# B&R Automation Studio project Panasonic_LinkaKapacitorov_A2021040 (part 6)

#### Main.st - Init, cyclic, exit code
```iecst
PROGRAM _INIT
	(* Insert code here *)

END_PROGRAM

PROGRAM _CYCLIC

	//Meranie motohodin ionizátora Tajfun//

	Tajfun_Motohodiny.START:= Linka.OUT.IonJednotka_START;

	//Spustenie merania//
	IF Tajfun_Motohodiny.START THEN
		Tajfun_Motohodiny.Milisekundy:= Tajfun_Motohodiny.Milisekundy + 2;//Ak je v taskovej triede 2ms tak prirátaváme + 2//
	END_IF

	IF Tajfun_Motohodiny.Milisekundy >= 1000 THEN
		Tajfun_Motohodiny.Sekundy:= Tajfun_Motohodiny.Sekundy + 1;
		Tajfun_Motohodiny.Milisekundy:= 0;
	END_IF

	IF Tajfun_Motohodiny.Sekundy >= 60 THEN
		Tajfun_Motohodiny.Minuty:= Tajfun_Motohodiny.Minuty + 1;
		Tajfun_Motohodiny.Sekundy:= 0;
	END_IF

	IF Tajfun_Motohodiny.Minuty >= 60 THEN
		Tajfun_Motohodiny.Hodiny:= Tajfun_Motohodiny.Hodiny + 1;
		Tajfun_Motohodiny.CelkovyPocetHodin:= Tajfun_Motohodiny.CelkovyPocetHodin + 1;
		Tajfun_Motohodiny.Minuty:= 0;
	END_IF

	IF Tajfun_Motohodiny.Hodiny >= 24 THEN
		Tajfun_Motohodiny.Dny:= Tajfun_Motohodiny.Dny + 1;
		Tajfun_Motohodiny.Hodiny:= 0;
	END_IF

	//Reset merania//
	IF Tajfun_Motohodiny.RESET THEN
		Tajfun_Motohodiny.Milisekundy:= 0;
		Tajfun_Motohodiny.Sekundy:= 0;
		Tajfun_Motohodiny.Minuty:= 0;
		Tajfun_Motohodiny.Hodiny:= 0;
		Tajfun_Motohodiny.CelkovyPocetHodin:= 0;
		Tajfun_Motohodiny.Dny:= 0;
		Tajfun_Motohodiny.RESET:= FALSE;
	END_IF

	//Zobrazenie stavov filtrov ionizačnej jednotky//
	//0 - Stav filtrov ionizačnej jednotky je OK.
	//1 - Blíži sa termín výmeny filtrov ionizačnej jednotky !!!
	//2 - Nutná výmena filtrov ionizačnej jednotky !!!

	//Farby stavov filtrov//
	//0 - Sivá
	//1 - Zelená
	//2 - Oranžová
	//3 - Červená

	CasKontrolyFiltrov.IN:= Linka.OUT.IonJednotka_START;

	IF Safety.STAV.SafetyPLC_Nabehlo THEN
		IF CasKontrolyFiltrov.Q AND (NOT Linka.IN.IonJednotka_Error_Filter1_RJ1 OR NOT Linka.IN.IonJednotka_Error_Filter2_RJ1)THEN
			Linka.STAV.FiltreIonizacnejJednotkyZanesene:= TRUE;
			Vizu.IndexStavuFiltrov:= 2;
			Vizu.IndexFarbyStavuFiltrov:= 3;
		ELSIF Tajfun_Motohodiny.Dny >= RemPremenne.PocetDniDoVymenyFiltra THEN
			Linka.STAV.FiltreIonizacnejJednotkyZanesene:= TRUE;
			Vizu.IndexStavuFiltrov:= 2;
			Vizu.IndexFarbyStavuFiltrov:= 3;
		ELSIF Tajfun_Motohodiny.Dny >= RemPremenne.PocetDniDoVymenyFiltra - 7 THEN
			Vizu.IndexStavuFiltrov:= 1;
			Vizu.IndexFarbyStavuFiltrov:= 2;
		ELSE
			Vizu.IndexStavuFiltrov:= 0;
			Vizu.IndexFarbyStavuFiltrov:= 1;
		END_IF
	END_IF

	IF Linka.VymenaFiltrovPotvrdena THEN
		Linka.STAV.FiltreIonizacnejJednotkyZanesene:= FALSE;
		Tajfun_Motohodiny.RESET:= TRUE;
		Linka.VymenaFiltrovPotvrdena:= FALSE;
	END_IF

	CasKontrolyFiltrov.PT:= T#2s;
	CasKontrolyFiltrov();

END_PROGRAM

PROGRAM _EXIT
	(* Insert code here *)

END_PROGRAM
```

#### Variables.var - Local variables
```iecst
VAR
	CasKontrolyFiltrov : TON := (0);
END_VAR
```

### Program Logical/Program/TestKomunikacie (IEC)

#### Main.st - Init, cyclic, exit code
```iecst
PROGRAM _INIT
	(* Insert code here *)

END_PROGRAM

PROGRAM _CYCLIC

	//Volanie funkcie SequenceControl//
	SequenceControl(SC:= SC_Step);

	CASE SC_Step.Step OF

		0:
			SC_Step.StepName:='0 - Nulovanie';
			Cistenie_OK:= FALSE;
			Cistenie_NG:= FALSE;
			VytlacEtiketu:= FALSE;
			NalepenieEtikety_OK:= FALSE;
			NalepenieEikety_NG:= FALSE;
			KontrolaDMkodu_OK:= FALSE;
			KontrolaDMkodu_NG:= FALSE;
			KontrolaTextu_OK:= FALSE;
			KontrolaTextu_NG:= FALSE;
			KOM_Panasonic.Server_IN.DataForServer_READY:= FALSE;
			KOM_Panasonic.Server_IN.ProcessResult:= FALSE;
			KOM_Panasonic.Server_IN.CommandNumber:= 0;
			SC_Step.ResetStep:= TRUE;
			SC_Step.Step:= 1;

		1:
			IF Cistenie_OK THEN
				ZakaznickeCislo:= '';
				ReturnProcessName:= '';
				SC_Step.ResetStep:= TRUE;
				SC_Step.Step:= 10;
			ELSIF Cistenie_NG THEN
				ZakaznickeCislo:= '';
				ReturnProcessName:= '';
				SC_Step.ResetStep:= TRUE;
				SC_Step.Step:= 20;
			ELSIF VytlacEtiketu THEN
				ReturnProcessName:= '';
				SC_Step.ResetStep:= TRUE;
				SC_Step.Step:= 30;
			ELSIF NalepenieEtikety_OK THEN
				ReturnProcessName:= '';
				SC_Step.ResetStep:= TRUE;
				SC_Step.Step:= 40;
			ELSIF NalepenieEikety_NG THEN
				ReturnProcessName:= '';
				SC_Step.ResetStep:= TRUE;
				SC_Step.Step:= 50;
			ELSIF KontrolaDMkodu_OK THEN
				ReturnProcessName:= '';
				SC_Step.ResetStep:= TRUE;
				SC_Step.Step:= 60;
			ELSIF KontrolaDMkodu_NG THEN
				ReturnProcessName:= '';
				SC_Step.ResetStep:= TRUE;
				SC_Step.Step:= 70;
			ELSIF KontrolaTextu_OK THEN
				ReturnProcessName:= '';
				SC_Step.ResetStep:= TRUE;
				SC_Step.Step:= 80;
			ELSIF KontrolaTextu_NG THEN
				ReturnProcessName:= '';
				SC_Step.ResetStep:= TRUE;
				SC_Step.Step:= 90;
			END_IF

		10:
			SC_Step.StepName:='10 - Odoslanie - Stav cistenie OK';
			SC_Step.IdleTime.PT:= T#4s;
			SC_Step.AlarmTime.PT:= T#5s;

			KOM_Panasonic.Server_IN.NazovPaletky_RFID:= '10_CP1';
			KOM_Panasonic.Server_IN.SerialNumber_InternaEtiketa:= 'BD10020070300046ZZZZZZZB10BD1';
			KOM_Panasonic.Server_IN.Cislo_LOTU:= 'BS217210002';

			IF NOT KOM_Panasonic.Server_OUT.DataForPLC_READY THEN
				KOM_Panasonic.Server_IN.CommandNumber:= 10;
				KOM_Panasonic.Server_IN.ProcessResult:= TRUE;
				KOM_Panasonic.Server_IN.DataForServer_READY:= TRUE;
				SC_Step.ResetStep:= TRUE;
				SC_Step.Step:= 13;
			END_IF

		13:
			SC_Step.StepName:='13 - Odpoved servera';
			SC_Step.IdleTime.PT:= T#100ms;
			SC_Step.AlarmTime.PT:= T#5s;

			IF KOM_Panasonic.Server_OUT.DataForPLC_READY AND KOM_Panasonic.Server_OUT.LastCommandNumber = 10 THEN
				IF KOM_Panasonic.Server_OUT.ContinueToNextProcess THEN
					ZakaznickeCislo:= KOM_Panasonic.Server_OUT.SerialNumber_ZakaznickaEtiketa;
					KOM_Panasonic.Server_IN.DataForServer_READY:= FALSE;
					ReturnProcessName:= 'OK';
					SC_Step.ResetStep:= TRUE;
					SC_Step.Step:= 0;
				ELSIF NOT KOM_Panasonic.Server_OUT.ContinueToNextProcess THEN
					ReturnProcessName:= KOM_Panasonic.Server_OUT.ReturnProcessName;
					KOM_Panasonic.Server_IN.DataForServer_READY:= FALSE;
					SC_Step.ResetStep:= TRUE;
					SC_Step.Step:= 0;
				END_IF
			END_IF

		20:
			SC_Step.StepName:='20 - Odoslanie - Stav cistenie NG';
			SC_Step.IdleTime.PT:= T#4s;
			SC_Step.AlarmTime.PT:= T#5s;

			KOM_Panasonic.Server_IN.NazovPaletky_RFID:= '10_CP1';
			KOM_Panasonic.Server_IN.SerialNumber_InternaEtiketa:= 'BD10020070300046ZZZZZZZB10BD1';
			KOM_Panasonic.Server_IN.Cislo_LOTU:= 'BS217210002';

			IF NOT KOM_Panasonic.Server_OUT.DataForPLC_READY THEN
				KOM_Panasonic.Server_IN.CommandNumber:= 10;
				KOM_Panasonic.Server_IN.ProcessResult:= FALSE;
				KOM_Panasonic.Server_IN.DataForServer_READY:= TRUE;
				SC_Step.ResetStep:= TRUE;
				SC_Step.Step:= 23;
			END_IF

		23:
			SC_Step.StepName:='23 - Odpoved servera';
			SC_Step.IdleTime.PT:= T#100ms;
			SC_Step.AlarmTime.PT:= T#5s;

			IF KOM_Panasonic.Server_OUT.DataForPLC_READY AND KOM_Panasonic.Server_OUT.LastCommandNumber = 10 THEN
				IF KOM_Panasonic.Server_OUT.ContinueToNextProcess THEN
					ZakaznickeCislo:= KOM_Panasonic.Server_OUT.SerialNumber_ZakaznickaEtiketa;
					KOM_Panasonic.Server_IN.DataForServer_READY:= FALSE;
					ReturnProcessName:= 'OK';
					SC_Step.ResetStep:= TRUE;
					SC_Step.Step:= 0;
				ELSIF NOT KOM_Panasonic.Server_OUT.ContinueToNextProcess THEN
					ReturnProcessName:= KOM_Panasonic.Server_OUT.ReturnProcessName;
					KOM_Panasonic.Server_IN.DataForServer_READY:= FALSE;
					SC_Step.ResetStep:= TRUE;
					SC_Step.Step:= 0;
				END_IF
			END_IF

		30:
			SC_Step.StepName:='30 - Odoslanie - Vytlac etiketu';
			SC_Step.IdleTime.PT:= T#4s;
			SC_Step.AlarmTime.PT:= T#5s;

			KOM_Panasonic.Server_IN.NazovPaletky_RFID:= '10_CP1';
			KOM_Panasonic.Server_IN.SerialNumber_InternaEtiketa:= 'BD10020070300046ZZZZZZZB10BD1';
			KOM_Panasonic.Server_IN.Cislo_LOTU:= 'BS217210002';

			IF NOT KOM_Panasonic.Server_OUT.DataForPLC_READY THEN
				KOM_Panasonic.Server_IN.CommandNumber:= 20;
				KOM_Panasonic.Server_IN.ProcessResult:= TRUE;
				KOM_Panasonic.Server_IN.DataForServer_READY:= TRUE;
				SC_Step.ResetStep:= TRUE;
				SC_Step.Step:= 33;
			END_IF

		33:
			SC_Step.StepName:='33 - Odpoved servera';
			SC_Step.IdleTime.PT:= T#100ms;
			SC_Step.AlarmTime.PT:= T#5s;

			IF KOM_Panasonic.Server_OUT.DataForPLC_READY AND KOM_Panasonic.Server_OUT.LastCommandNumber = 20 THEN
				IF KOM_Panasonic.Server_OUT.ContinueToNextProcess THEN
					KOM_Panasonic.Server_IN.DataForServer_READY:= FALSE;
					ReturnProcessName:= 'OK';
					SC_Step.ResetStep:= TRUE;
					SC_Step.Step:= 0;
				ELSIF NOT KOM_Panasonic.Server_OUT.ContinueToNextProcess THEN
					ReturnProcessName:= KOM_Panasonic.Server_OUT.ReturnProcessName;
					KOM_Panasonic.Server_IN.DataForServer_READY:= FALSE;
					SC_Step.ResetStep:= TRUE;
					SC_Step.Step:= 0;
				END_IF
			END_IF

		40:
			SC_Step.StepName:='40 - Odoslanie - Stav nalepenie etikety OK';
			SC_Step.IdleTime.PT:= T#4s;
			SC_Step.AlarmTime.PT:= T#5s;

			KOM_Panasonic.Server_IN.NazovPaletky_RFID:= '10_CP1';
			KOM_Panasonic.Server_IN.SerialNumber_InternaEtiketa:= 'BD10020070300046ZZZZZZZB10BD1';
			KOM_Panasonic.Server_IN.Cislo_LOTU:= 'BS217210002';

			IF NOT KOM_Panasonic.Server_OUT.DataForPLC_READY THEN
				KOM_Panasonic.Server_IN.CommandNumber:= 30;
				KOM_Panasonic.Server_IN.ProcessResult:= TRUE;
				KOM_Panasonic.Server_IN.DataForServer_READY:= TRUE;
				SC_Step.ResetStep:= TRUE;
				SC_Step.Step:= 43;
			END_IF

		43:
			SC_Step.StepName:='43 - Odpoved servera';
			SC_Step.IdleTime.PT:= T#100ms;
			SC_Step.AlarmTime.PT:= T#5s;

			IF KOM_Panasonic.Server_OUT.DataForPLC_READY AND KOM_Panasonic.Server_OUT.LastCommandNumber = 30 THEN
				IF KOM_Panasonic.Server_OUT.ContinueToNextProcess THEN
					KOM_Panasonic.Server_IN.DataForServer_READY:= FALSE;
					ReturnProcessName:= 'OK';
					SC_Step.ResetStep:= TRUE;
					SC_Step.Step:= 0;
				ELSIF NOT KOM_Panasonic.Server_OUT.ContinueToNextProcess THEN
					ReturnProcessName:= KOM_Panasonic.Server_OUT.ReturnProcessName;
					KOM_Panasonic.Server_IN.DataForServer_READY:= FALSE;
					SC_Step.ResetStep:= TRUE;
					SC_Step.Step:= 0;
				END_IF
			END_IF

		50:
			SC_Step.StepName:='50 - Odoslanie - Stav nalepenie etikety NG';
			SC_Step.IdleTime.PT:= T#4s;
			SC_Step.AlarmTime.PT:= T#5s;

			KOM_Panasonic.Server_IN.NazovPaletky_RFID:= '10_CP1';
			KOM_Panasonic.Server_IN.SerialNumber_InternaEtiketa:= 'BD10020070300046ZZZZZZZB10BD1';
			KOM_Panasonic.Server_IN.Cislo_LOTU:= 'BS217210002';

			IF NOT KOM_Panasonic.Server_OUT.DataForPLC_READY THEN
				KOM_Panasonic.Server_IN.CommandNumber:= 30;
				KOM_Panasonic.Server_IN.ProcessResult:= FALSE;
				KOM_Panasonic.Server_IN.DataForServer_READY:= TRUE;
				SC_Step.ResetStep:= TRUE;
				SC_Step.Step:= 53;
			END_IF

		53:
			SC_Step.StepName:='53 - Odpoved servera';
			SC_Step.IdleTime.PT:= T#100ms;
			SC_Step.AlarmTime.PT:= T#5s;

			IF KOM_Panasonic.Server_OUT.DataForPLC_READY AND KOM_Panasonic.Server_OUT.LastCommandNumber = 30 THEN
				IF KOM_Panasonic.Server_OUT.ContinueToNextProcess THEN
					KOM_Panasonic.Server_IN.DataForServer_READY:= FALSE;
					ReturnProcessName:= 'OK';
					SC_Step.ResetStep:= TRUE;
					SC_Step.Step:= 0;
				ELSIF NOT KOM_Panasonic.Server_OUT.ContinueToNextProcess THEN
					ReturnProcessName:= KOM_Panasonic.Server_OUT.ReturnProcessName;
					KOM_Panasonic.Server_IN.DataForServer_READY:= FALSE;
					SC_Step.ResetStep:= TRUE;
					SC_Step.Step:= 0;
				END_IF
			END_IF

		60:
			SC_Step.StepName:='60 - Odoslanie - Stav citania DM kodu zakaznickej etikety OK';
			SC_Step.IdleTime.PT:= T#4s;
			SC_Step.AlarmTime.PT:= T#5s;

			KOM_Panasonic.Server_IN.NazovPaletky_RFID:= '10_CP1';
			KOM_Panasonic.Server_IN.SerialNumber_InternaEtiketa:= 'BD10020070300046ZZZZZZZB10BD1';
			KOM_Panasonic.Server_IN.Cislo_LOTU:= 'BS217210002';

			IF NOT KOM_Panasonic.Server_OUT.DataForPLC_READY THEN
				KOM_Panasonic.Server_IN.CommandNumber:= 40;
				KOM_Panasonic.Server_IN.ProcessResult:= TRUE;
				KOM_Panasonic.Server_IN.DataForServer_READY:= TRUE;
				SC_Step.ResetStep:= TRUE;
				SC_Step.Step:= 63;
			END_IF

		63:
			SC_Step.StepName:='63 - Odpoved servera';
			SC_Step.IdleTime.PT:= T#100ms;
			SC_Step.AlarmTime.PT:= T#5s;

			IF KOM_Panasonic.Server_OUT.DataForPLC_READY AND KOM_Panasonic.Server_OUT.LastCommandNumber = 40 THEN
				IF KOM_Panasonic.Server_OUT.ContinueToNextProcess THEN
					KOM_Panasonic.Server_IN.DataForServer_READY:= FALSE;
					ReturnProcessName:= 'OK';
					SC_Step.ResetStep:= TRUE;
					SC_Step.Step:= 0;
				ELSIF NOT KOM_Panasonic.Server_OUT.ContinueToNextProcess THEN
					ReturnProcessName:= KOM_Panasonic.Server_OUT.ReturnProcessName;
					KOM_Panasonic.Server_IN.DataForServer_READY:= FALSE;
					SC_Step.ResetStep:= TRUE;
					SC_Step.Step:= 0;
				END_IF
			END_IF

		70:
			SC_Step.StepName:='70 - Odoslanie - Stav citania DM kodu zakaznickej etikety NG';
			SC_Step.IdleTime.PT:= T#4s;
			SC_Step.AlarmTime.PT:= T#5s;

			KOM_Panasonic.Server_IN.NazovPaletky_RFID:= '10_CP1';
			KOM_Panasonic.Server_IN.SerialNumber_InternaEtiketa:= 'BD10020070300046ZZZZZZZB10BD1';
			KOM_Panasonic.Server_IN.Cislo_LOTU:= 'BS217210002';

			IF NOT KOM_Panasonic.Server_OUT.DataForPLC_READY THEN
				KOM_Panasonic.Server_IN.CommandNumber:= 40;
				KOM_Panasonic.Server_IN.ProcessResult:= FALSE;
				KOM_Panasonic.Server_IN.DataForServer_READY:= TRUE;
				SC_Step.ResetStep:= TRUE;
				SC_Step.Step:= 73;
			END_IF

		73:
			SC_Step.StepName:='73 - Odpoved servera';
			SC_Step.IdleTime.PT:= T#100ms;
			SC_Step.AlarmTime.PT:= T#5s;

			IF KOM_Panasonic.Server_OUT.DataForPLC_READY AND KOM_Panasonic.Server_OUT.LastCommandNumber = 40 THEN
				IF KOM_Panasonic.Server_OUT.ContinueToNextProcess THEN
					KOM_Panasonic.Server_IN.DataForServer_READY:= FALSE;
					ReturnProcessName:= 'OK';
					SC_Step.ResetStep:= TRUE;
					SC_Step.Step:= 0;
				ELSIF NOT KOM_Panasonic.Server_OUT.ContinueToNextProcess THEN
					ReturnProcessName:= KOM_Panasonic.Server_OUT.ReturnProcessName;
					KOM_Panasonic.Server_IN.DataForServer_READY:= FALSE;
					SC_Step.ResetStep:= TRUE;
					SC_Step.Step:= 0;
				END_IF
			END_IF

		80:
			SC_Step.StepName:='80 - Odoslanie - Stav citania znakov zakaznickej etikety OK';
			SC_Step.IdleTime.PT:= T#4s;
			SC_Step.AlarmTime.PT:= T#5s;

			KOM_Panasonic.Server_IN.NazovPaletky_RFID:= '10_CP1';
			KOM_Panasonic.Server_IN.SerialNumber_InternaEtiketa:= 'BD10020070300046ZZZZZZZB10BD1';
			KOM_Panasonic.Server_IN.Cislo_LOTU:= 'BS217210002';

			IF NOT KOM_Panasonic.Server_OUT.DataForPLC_READY THEN
				KOM_Panasonic.Server_IN.CommandNumber:= 50;
				KOM_Panasonic.Server_IN.ProcessResult:= TRUE;
				KOM_Panasonic.Server_IN.DataForServer_READY:= TRUE;
				SC_Step.ResetStep:= TRUE;
				SC_Step.Step:= 83;
			END_IF

		83:
			SC_Step.StepName:='83 - Odpoved servera';
			SC_Step.IdleTime.PT:= T#100ms;
			SC_Step.AlarmTime.PT:= T#5s;

			IF KOM_Panasonic.Server_OUT.DataForPLC_READY AND KOM_Panasonic.Server_OUT.LastCommandNumber = 50 THEN
				IF KOM_Panasonic.Server_OUT.ContinueToNextProcess THEN
					KOM_Panasonic.Server_IN.DataForServer_READY:= FALSE;
					ReturnProcessName:= 'OK';
					SC_Step.ResetStep:= TRUE;
					SC_Step.Step:= 0;
				ELSIF NOT KOM_Panasonic.Server_OUT.ContinueToNextProcess THEN
					ReturnProcessName:= KOM_Panasonic.Server_OUT.ReturnProcessName;
					KOM_Panasonic.Server_IN.DataForServer_READY:= FALSE;
					SC_Step.ResetStep:= TRUE;
					SC_Step.Step:= 0;
				END_IF
			END_IF

		90:
			SC_Step.StepName:='90 - Odoslanie - Stav citania znakov zakaznickej etikety NG';
			SC_Step.IdleTime.PT:= T#4s;
			SC_Step.AlarmTime.PT:= T#5s;

			KOM_Panasonic.Server_IN.NazovPaletky_RFID:= '10_CP1';
			KOM_Panasonic.Server_IN.SerialNumber_InternaEtiketa:= 'BD10020070300046ZZZZZZZB10BD1';
			KOM_Panasonic.Server_IN.Cislo_LOTU:= 'BS217210002';

			IF NOT KOM_Panasonic.Server_OUT.DataForPLC_READY THEN
				KOM_Panasonic.Server_IN.CommandNumber:= 50;
				KOM_Panasonic.Server_IN.ProcessResult:= FALSE;
				KOM_Panasonic.Server_IN.DataForServer_READY:= TRUE;
				SC_Step.ResetStep:= TRUE;
				SC_Step.Step:= 93;
			END_IF

		93:
			SC_Step.StepName:='93 - Odpoved servera';
			SC_Step.IdleTime.PT:= T#100ms;
			SC_Step.AlarmTime.PT:= T#5s;

			IF KOM_Panasonic.Server_OUT.DataForPLC_READY AND KOM_Panasonic.Server_OUT.LastCommandNumber = 50 THEN
				IF KOM_Panasonic.Server_OUT.ContinueToNextProcess THEN
					KOM_Panasonic.Server_IN.DataForServer_READY:= FALSE;
					ReturnProcessName:= 'OK';
					SC_Step.ResetStep:= TRUE;
					SC_Step.Step:= 0;
				ELSIF NOT KOM_Panasonic.Server_OUT.ContinueToNextProcess THEN
					ReturnProcessName:= KOM_Panasonic.Server_OUT.ReturnProcessName;
					KOM_Panasonic.Server_IN.DataForServer_READY:= FALSE;
					SC_Step.ResetStep:= TRUE;
					SC_Step.Step:= 0;
				END_IF
			END_IF

	END_CASE

END_PROGRAM

PROGRAM _EXIT
	(* Insert code here *)

END_PROGRAM
```

#### Variables.var - Local variables
```iecst
VAR
	SC_Step : SequenceControlTyp := (0);
	Cistenie_OK : BOOL := 0;
	Cistenie_NG : BOOL := 0;
	VytlacEtiketu : BOOL := 0;
	NalepenieEtikety_OK : BOOL := 0;
	NalepenieEikety_NG : BOOL := 0;
	KontrolaDMkodu_OK : BOOL := 0;
	KontrolaDMkodu_NG : BOOL := 0;
	KontrolaTextu_OK : BOOL := 0;
	KontrolaTextu_NG : BOOL := 0;
	ZakaznickeCislo : STRING[49] := '';
	ReturnProcessName : STRING[80] := '0';
END_VAR
```

### Program Logical/HMI/OvladanieVizu (IEC)

#### Main.st - Init, cyclic, exit code
```iecst
PROGRAM _INIT
	Vizu.NacitanieLOTU_DISABLE:= TRUE;
	Vizu.ZobrazHlasenie_PotvrdPaletkyNG:= 1;
	Vizu.ZobrazHlasenie_NespravTypPaletky:= 1;
	Vizu.ZobrazHlasenie_ZaaretujTlaciaren:= 1;
	Vizu.ZobrazHlas_ZatvorSerDvereTlac:= 1;
	Vizu.ZobrazHlasenie_TlaciarenOffline:= 1;
	Vizu.ZobrazHlasenie_DochadzaPaska:= 1;
END_PROGRAM

PROGRAM _CYCLIC

	//Prepnutie na hlavnu obrazovku pri stlačení tlačítka CS//
	IF EDGENEG(Safety.STAV.ZonaCS_AKTIVNA)THEN
		Vizu.CisloZadanejObrazovky:= 2;
	END_IF

	//Zmena jazyka vizualizácie//
	Vizu.Language_Index;

	//**********************************************Urovne uživatelov***********************************************************//
	//10 - Zoraďovač
	//20 - Zvláštna uroveň
	//30 - Technológ
	//40 - Admin Technológ

	//***********************************************Zobrazenie stavov zariadenia***********************************************//
    //0 - Linka je vypnutá.
    //1 - Prebieha inicializacia linky.
    //2 - Linka beží v automatickom režime.
    //3 - Robot nieje prepnutý do automatického režimu !!!
	//4 - Prebieha ukoncenie cyklu.
    //5 - Nieje zvolený model alebo LOT !!!
	//6 - Tlačiareň nieje Online !!!
	//7 - Tlačiareň nieje zaistená !!!
	//8 - Servisné dvere tlačiarne niesu zatvorené !!!
	//9 - Paletka sa nachádza v bariere dopravnika NG !!!
	//10 - V tlačiarni došli etikety !!!
	//11 - V tlačiarni došla termopáska !!!
	//12 - Filtre ionizačnej jednotky sú zanesené !!!
	//13 - Kamera robota nieje READY !!!
	//14 - Dvere bunky niesu zamknuté !!!

	IF NOT Robot.KOM_IN.Stav_RezimAUTOMAT THEN
		Vizu.StavZariadenia_Index:= 3;
		Vizu.StavZariadenia_Farba:= 3;
	ELSIF Linka.PAR.Zvoleny_MODEL = '' OR Linka.PAR.Zvoleny_LOT = '' THEN
		Vizu.StavZariadenia_Index:= 5;
		Vizu.StavZariadenia_Farba:= 3;
	ELSIF StoperEtiketovania.IN.Tlaciaren_Offline THEN
		Vizu.StavZariadenia_Index:= 6;
		Vizu.StavZariadenia_Farba:= 3;
	ELSIF NOT StoperEtiketovania.STAV.TlaciarenZaaretovana THEN
		Vizu.StavZariadenia_Index:= 7;
		Vizu.StavZariadenia_Farba:= 3;
	ELSIF NOT Robot.Automat AND NOT Safety.STAV.BarieraDopravnikaNG_AKTIVNA THEN
		Vizu.StavZariadenia_Index:= 9;
		Vizu.StavZariadenia_Farba:= 3;
	ELSIF NOT Safety.STAV.ServisneDvereTlaciarne_AKTIVNE THEN
		Vizu.StavZariadenia_Index:= 8;
		Vizu.StavZariadenia_Farba:= 3;
	ELSIF StoperEtiketovania.IN.Tlaciaren_KoniecEtikiet THEN
		Vizu.StavZariadenia_Index:= 10;
		Vizu.StavZariadenia_Farba:= 3;
	ELSIF StoperEtiketovania.IN.Tlaciaren_KoniecPasky THEN
		Vizu.StavZariadenia_Index:= 11;
		Vizu.StavZariadenia_Farba:= 3;
	ELSIF Linka.STAV.FiltreIonizacnejJednotkyZanesene THEN
		Vizu.StavZariadenia_Index:= 12;
		Vizu.StavZariadenia_Farba:= 3;
	ELSIF NOT Kamera.STAV.READY THEN
		Vizu.StavZariadenia_Index:= 13;
		Vizu.StavZariadenia_Farba:= 3;
	ELSIF NOT Safety.STAV.ZonaBunky_AKTIVNA THEN
		Vizu.StavZariadenia_Index:= 14;
		Vizu.StavZariadenia_Farba:= 3;
	ELSIF Linka.STAV.Automat AND Linka.STAV.UkoncenieCyklu_BUSY THEN
		Vizu.StavZariadenia_Index:= 4;
		Vizu.StavZariadenia_Farba:= 4;
	ELSIF Linka.STAV.Automat AND NOT Linka.STAV.PoINIT THEN
		Vizu.StavZariadenia_Index:= 1;
		Vizu.StavZariadenia_Farba:= 1;
	ELSIF Linka.STAV.Automat AND Linka.STAV.PoINIT THEN
		Vizu.StavZariadenia_Index:= 2;
		Vizu.StavZariadenia_Farba:= 2;
	ELSE
		Vizu.StavZariadenia_Index:= 0;
		Vizu.StavZariadenia_Farba:= 0;
	END_IF

	//******************************************************Podsvietenie tlačítok**********************************************************//

	//Tlačítko alarmy//
	IF NastalaPorucha THEN
		Vizu.FarbaTlacitkaAlarm_Index:= Blikac500ms;
	ELSE
		Vizu.FarbaTlacitkaAlarm_Index:= FALSE;
	END_IF

	//Zobrazenie symbolov stlačeného CS//
	IF Safety.STAV.CS_VstupnyVytah_Odblokovany THEN
		Vizu.ZobrazSymbolCS_VstupVytah:= 1;
	ELSE
		Vizu.ZobrazSymbolCS_VstupVytah:= 0;
	END_IF

	IF Safety.STAV.CS_VystupnyVytah_Odblokovany THEN
		Vizu.ZobrazSymbolCS_VystupVytah:= 1;
	ELSE
		Vizu.ZobrazSymbolCS_VystupVytah:= 0;
	END_IF

	IF Safety.STAV.CS_OvlPanel_Odblokovany THEN
		Vizu.ZobrazSymbolCS_Panel:= 1;
	ELSE
		Vizu.ZobrazSymbolCS_Panel:= 0;
	END_IF

	IF Safety.STAV.CS_Robot_Odblokovany THEN
		Vizu.ZobrazSymbolCS_Robot:= 1;
	ELSE
		Vizu.ZobrazSymbolCS_Robot:= 0;
	END_IF

	//**********************************************Zobrazenie stavov jednotlivých pracovisk****************************************//
	//Vstupny výtah//
	IF VstupVytah.Automat AND VstupVytah.KoniecCyklu THEN
		Vizu.StavPracoviskaVstupVytah_Index:= 4;
	ELSIF VstupVytah.Automat AND NOT VstupVytah.STAV.PoINIT THEN
		Vizu.StavPracoviskaVstupVytah_Index:= 1;
	ELSIF VstupVytah.Automat AND VstupVytah.STAV.PoINIT THEN
		Vizu.StavPracoviskaVstupVytah_Index:= 2;
	ELSE
		Vizu.StavPracoviskaVstupVytah_Index:= 0;
	END_IF

	//Stoper pred čistením//
	IF StoperPredCistenim.Automat AND StoperPredCistenim.KoniecCyklu THEN
		Vizu.StavPracoviskaStopPredCist_Index:= 4;
	ELSIF StoperPredCistenim.Automat AND NOT StoperPredCistenim.STAV.PoINIT THEN
		Vizu.StavPracoviskaStopPredCist_Index:= 1;
	ELSIF StoperPredCistenim.Automat AND StoperPredCistenim.STAV.PoINIT THEN
		Vizu.StavPracoviskaStopPredCist_Index:= 2;
	ELSE
		Vizu.StavPracoviskaStopPredCist_Index:= 0;
	END_IF

	//Stoper po čistení//
	IF StoperPoCisteni.Automat AND StoperPoCisteni.KoniecCyklu THEN
		Vizu.StavPracoviskaStopPoCist_Index:= 4;
	ELSIF StoperPoCisteni.Automat AND NOT StoperPoCisteni.STAV.PoINIT THEN
		Vizu.StavPracoviskaStopPoCist_Index:= 1;
	ELSIF StoperPoCisteni.Automat AND StoperPoCisteni.STAV.PoINIT THEN
		Vizu.StavPracoviskaStopPoCist_Index:= 2;
	ELSE
		Vizu.StavPracoviskaStopPoCist_Index:= 0;
	END_IF

	//Dopravník čistenia//
	IF DopravCistenia.Automat AND DopravCistenia.KoniecCyklu THEN
		Vizu.StavPracoviskaDoprCistenia_Index:= 4;
	ELSIF DopravCistenia.Automat AND NOT DopravCistenia.STAV.PoINIT THEN
		Vizu.StavPracoviskaDoprCistenia_Index:= 1;
	ELSIF DopravCistenia.Automat AND DopravCistenia.STAV.PoINIT THEN
		Vizu.StavPracoviskaDoprCistenia_Index:= 2;
	ELSE
		Vizu.StavPracoviskaDoprCistenia_Index:= 0;
	END_IF

	//Stoper etiketovania//
	IF StoperEtiketovania.Automat AND StoperEtiketovania.KoniecCyklu THEN
		Vizu.StavPracoviskaStopEtiketov_Index:= 4;
	ELSIF StoperEtiketovania.Automat AND NOT StoperEtiketovania.STAV.PoINIT THEN
		Vizu.StavPracoviskaStopEtiketov_Index:= 1;
	ELSIF StoperEtiketovania.Automat AND StoperEtiketovania.STAV.PoINIT THEN
		Vizu.StavPracoviskaStopEtiketov_Index:= 2;
	ELSE
		Vizu.StavPracoviskaStopEtiketov_Index:= 0;
	END_IF

	//Robot//
	IF Robot.Automat AND Robot.KoniecCyklu THEN
		Vizu.StavPracoviskaRobota_Index:= 4;
	ELSIF Robot.Automat AND NOT Robot.STAV.PoINIT THEN
		Vizu.StavPracoviskaRobota_Index:= 1;
	ELSIF Robot.Automat AND Robot.STAV.PoINIT THEN
		Vizu.StavPracoviskaRobota_Index:= 2;
	ELSE
		Vizu.StavPracoviskaRobota_Index:= 0;
	END_IF

	//Stoper dopravníka NG//
	IF StoperDopravNG.Automat AND StoperDopravNG.KoniecCyklu THEN
		Vizu.StavPracoviskaStopDopNG_Index:= 4;
	ELSIF StoperDopravNG.Automat AND NOT StoperDopravNG.STAV.PoINIT THEN
		Vizu.StavPracoviskaStopDopNG_Index:= 1;
	ELSIF StoperDopravNG.Automat AND StoperDopravNG.STAV.PoINIT THEN
		Vizu.StavPracoviskaStopDopNG_Index:= 2;
	ELSE
		Vizu.StavPracoviskaStopDopNG_Index:= 0;
	END_IF

	//Dopravník bunky//
	IF DopravBunky.Automat AND DopravBunky.KoniecCyklu THEN
		Vizu.StavPracoviskaDoprBunky_Index:= 4;
	ELSIF DopravBunky.Automat AND NOT DopravBunky.STAV.PoINIT THEN
		Vizu.StavPracoviskaDoprBunky_Index:= 1;
	ELSIF DopravBunky.Automat AND DopravBunky.STAV.PoINIT THEN
		Vizu.StavPracoviskaDoprBunky_Index:= 2;
	ELSE
		Vizu.StavPracoviskaDoprBunky_Index:= 0;
	END_IF

	//Stoper výstupného dopravníka//
	IF StoperVystupDopravnika.Automat AND StoperVystupDopravnika.KoniecCyklu THEN
		Vizu.StavPracoviskaStopVystDopr_Index:= 4;
	ELSIF StoperVystupDopravnika.Automat AND NOT StoperVystupDopravnika.STAV.PoINIT THEN
		Vizu.StavPracoviskaStopVystDopr_Index:= 1;
	ELSIF StoperVystupDopravnika.Automat AND StoperVystupDopravnika.STAV.PoINIT THEN
		Vizu.StavPracoviskaStopVystDopr_Index:= 2;
	ELSE
		Vizu.StavPracoviskaStopVystDopr_Index:= 0;
	END_IF

	//Výstupný dopravník//
	IF VystupnyDopravnik.Automat AND VystupnyDopravnik.KoniecCyklu THEN
		Vizu.StavPracoviskaDoprVystup_Index:= 4;
	ELSIF VystupnyDopravnik.Automat AND NOT VystupnyDopravnik.STAV.PoINIT THEN
		Vizu.StavPracoviskaDoprVystup_Index:= 1;
	ELSIF VystupnyDopravnik.Automat AND VystupnyDopravnik.STAV.PoINIT THEN
		Vizu.StavPracoviskaDoprVystup_Index:= 2;
	ELSE
		Vizu.StavPracoviskaDoprVystup_Index:= 0;
	END_IF

	//Výstupny výtah//
	IF VystupVytah.Automat AND VystupVytah.KoniecCyklu THEN
		Vizu.StavPracoviskaVystupVytah_Index:= 4;
	ELSIF VystupVytah.Automat AND NOT VystupVytah.STAV.PoINIT THEN
		Vizu.StavPracoviskaVystupVytah_Index:= 1;
	ELSIF VystupVytah.Automat AND VystupVytah.STAV.PoINIT THEN
		Vizu.StavPracoviskaVystupVytah_Index:= 2;
	ELSE
		Vizu.StavPracoviskaVystupVytah_Index:= 0;
	END_IF

	//Stoper vratného dopravníka//
	IF StoperVratDopravnika.Automat AND StoperVratDopravnika.KoniecCyklu THEN
		Vizu.StavPracoviskaStopVratDopr_Index:= 4;
	ELSIF StoperVratDopravnika.Automat AND NOT StoperVratDopravnika.STAV.PoINIT THEN
		Vizu.StavPracoviskaStopVratDopr_Index:= 1;
	ELSIF StoperVratDopravnika.Automat AND StoperVratDopravnika.STAV.PoINIT THEN
		Vizu.StavPracoviskaStopVratDopr_Index:= 2;
	ELSE
		Vizu.StavPracoviskaStopVratDopr_Index:= 0;
	END_IF

	//Vratný dopravník//
	IF VratnyDopravnik.Automat AND VratnyDopravnik.KoniecCyklu THEN
		Vizu.StavPracoviskaDoprVrat_Index:= 4;
	ELSIF VratnyDopravnik.Automat AND NOT VratnyDopravnik.STAV.PoINIT THEN
		Vizu.StavPracoviskaDoprVrat_Index:= 1;
	ELSIF VratnyDopravnik.Automat AND VratnyDopravnik.STAV.PoINIT THEN
		Vizu.StavPracoviskaDoprVrat_Index:= 2;
	ELSE
		Vizu.StavPracoviskaDoprVrat_Index:= 0;
	END_IF

	//*********************************************Zobrazenie úvodnej obrazovky**********************************************//
	IF NOT Safety.STAV.SafetyPLC_Nabehlo THEN
		Vizu.CisloZadanejObrazovky:= 0;
		IF EDGEPOS (Blikac500ms = TRUE) THEN
			IF Vizu.Slider < 30 THEN
				Vizu.Slider:= Vizu.Slider+1;
			ELSE
				Vizu.Slider:= 0;
			END_IF
		END_IF
	END_IF

	//************************************Prepnutie na obrazovku Automatického režimu******************************************//
	IF EDGEPOS (Safety.STAV.SafetyPLC_Nabehlo) THEN
		Vizu.CisloZadanejObrazovky:= 2;
	END_IF

	//*************************************************Zamknutie tlačítok*******************************************************//
	//Tlačítko režim manual//
	IF Linka.STAV.Automat THEN
		Vizu.TL_RezimManual_DISABLE:= TRUE;
	ELSIF NOT Safety.STAV.ZonaCS_AKTIVNA THEN
		Vizu.TL_RezimManual_DISABLE:= TRUE;
	ELSE
		Vizu.TL_RezimManual_DISABLE:= FALSE;
	END_IF

	//Tlačítko Štart Automat//
	IF NOT Safety.STAV.ZonaCS_AKTIVNA THEN
		Vizu.TL_StartAutomat_DISABLE:= TRUE;
	ELSIF NastalaPorucha THEN
		Vizu.TL_StartAutomat_DISABLE:= TRUE;
	ELSIF NOT Linka.STAV.Hardware_OK THEN
		Vizu.TL_StartAutomat_DISABLE:= TRUE;
	ELSIF Linka.PAR.Zvoleny_MODEL = '' THEN
		Vizu.TL_StartAutomat_DISABLE:= TRUE;
	ELSIF Linka.PAR.Zvoleny_LOT = '' THEN
		Vizu.TL_StartAutomat_DISABLE:= TRUE;
	ELSIF StoperEtiketovania.IN.Tlaciaren_Offline THEN
		Vizu.TL_StartAutomat_DISABLE:= TRUE;
	ELSIF NOT Robot.KOM_IN.Stav_RezimAUTOMAT THEN
		Vizu.TL_StartAutomat_DISABLE:= TRUE;
	ELSIF NOT StoperEtiketovania.STAV.TlaciarenZaaretovana THEN
		Vizu.TL_StartAutomat_DISABLE:= TRUE;
	ELSIF NOT Safety.STAV.ServisneDvereTlaciarne_AKTIVNE THEN
		Vizu.TL_StartAutomat_DISABLE:= TRUE;
	ELSIF NOT Robot.Automat AND NOT Safety.STAV.BarieraDopravnikaNG_AKTIVNA	THEN
		Vizu.TL_StartAutomat_DISABLE:= TRUE;
	ELSIF Linka.STAV.FiltreIonizacnejJednotkyZanesene THEN
		Vizu.TL_StartAutomat_DISABLE:= TRUE;
	ELSIF StoperEtiketovania.IN.Tlaciaren_KoniecEtikiet THEN
		Vizu.TL_StartAutomat_DISABLE:= TRUE;
	ELSIF StoperEtiketovania.IN.Tlaciaren_KoniecPasky THEN
		Vizu.TL_StartAutomat_DISABLE:= TRUE;
	ELSIF NOT Kamera.STAV.READY THEN
		Vizu.TL_StartAutomat_DISABLE:= TRUE;
	ELSIF NOT Safety.STAV.ZonaBunky_AKTIVNA THEN
		Vizu.TL_StartAutomat_DISABLE:= TRUE;
	ELSIF Linka.STAV.PoINIT THEN
		Vizu.TL_StartAutomat_DISABLE:= TRUE;
	ELSE
		Vizu.TL_StartAutomat_DISABLE:= FALSE;
	END_IF

	//Tlačítko Ukončenie cyklu//
	IF Linka.STAV.PoINIT THEN
		Vizu.TL_UkoncenieCyklu_DISABLE:= FALSE;
	ELSE
		Vizu.TL_UkoncenieCyklu_DISABLE:= TRUE;
	END_IF

	//Tlačítko Reset//
	IF Linka.STAV.PoINIT AND NOT Linka.STAV.UkoncenieCyklu_BUSY THEN
		Vizu.TL_Reset_DISABLE:= TRUE;
	ELSE
		Vizu.TL_Reset_DISABLE:= FALSE;
	END_IF

	//Zamknutie tlačítok ovládania zámkov dverí//
	IF Linka.STAV.Automat THEN
		Vizu.TL_ZamokPredneDvere_DISABLE:= TRUE;
		Vizu.TL_ZamokZadneDvere_DISABLE:= TRUE;
	ELSE
		Vizu.TL_ZamokPredneDvere_DISABLE:= FALSE;
		Vizu.TL_ZamokZadneDvere_DISABLE:= FALSE;
	END_IF

	//Tlačítko zmena modelu//
	IF Vizu.Nacitany_MODEL = '' THEN
		Vizu.TL_ZmenModel_DISABLE:= TRUE;
	ELSIF Vizu.Nacitany_LOT	= '' THEN
		Vizu.TL_ZmenModel_DISABLE:= TRUE;
	ELSE
		Vizu.TL_ZmenModel_DISABLE:= FALSE;
	END_IF

	//Tlačítko Homing vstupného výťahu//
	IF NOT Safety.STAV.ZonaVstupnyVytah_AKTIVNA THEN
		Vizu.TL_VstupVytah_Homing_DISABLE:= TRUE;
	ELSIF VstupVytah.STAV.Zdvih_BUSY THEN
		Vizu.TL_VstupVytah_Homing_DISABLE:= TRUE;
	ELSIF VstupVytah.RR_Dopravnik_VPRED THEN
		Vizu.TL_VstupVytah_Homing_DISABLE:= TRUE;
	ELSIF VstupVytah.RR_Dopravnik_VZAD THEN
		Vizu.TL_VstupVytah_Homing_DISABLE:= TRUE;
	ELSIF VstupVytah.IN.PrechodDopravnikaVytahu_OS1 THEN
		Vizu.TL_VstupVytah_Homing_DISABLE:= TRUE;
	ELSIF NOT VstupVytah.MenicZdvihu_FM2.STAV.READY THEN
		Vizu.TL_VstupVytah_Homing_DISABLE:= TRUE;
	ELSE
		Vizu.TL_VstupVytah_Homing_DISABLE:= FALSE;
	END_IF

	//Tlačítka zdvihu vstupného výťahu//
	IF NOT Safety.STAV.ZonaVstupnyVytah_AKTIVNA THEN
		Vizu.TL_VstupVytah_Zdvih_DISABLE:= TRUE;
	ELSIF VstupVytah.RR_Dopravnik_VPRED THEN
		Vizu.TL_VstupVytah_Zdvih_DISABLE:= TRUE;
	ELSIF VstupVytah.RR_Dopravnik_VZAD THEN
		Vizu.TL_VstupVytah_Zdvih_DISABLE:= TRUE;
	ELSIF VstupVytah.STAV.Homing_BUSY THEN
		Vizu.TL_VstupVytah_Zdvih_DISABLE:= TRUE;
	ELSIF VstupVytah.IN.PrechodDopravnikaVytahu_OS1 THEN
		Vizu.TL_VstupVytah_Zdvih_DISABLE:= TRUE;
	ELSIF NOT VstupVytah.MenicZdvihu_FM2.STAV.READY THEN
		Vizu.TL_VstupVytah_Zdvih_DISABLE:= TRUE;
	ELSE
		Vizu.TL_VstupVytah_Zdvih_DISABLE:= FALSE;
	END_IF

	//Tlačítko Homing vystupneho výťahu//
	IF NOT Safety.STAV.ZonaVystupnyVytah_AKTIVNA THEN
		Vizu.TL_VystupVytah_Homing_DISABLE:= TRUE;
	ELSIF VystupVytah.STAV.Zdvih_BUSY THEN
		Vizu.TL_VystupVytah_Homing_DISABLE:= TRUE;
	ELSIF VystupVytah.RR_Dopravnik_VPRED THEN
		Vizu.TL_VystupVytah_Homing_DISABLE:= TRUE;
	ELSIF VystupVytah.RR_Dopravnik_VZAD THEN
		Vizu.TL_VystupVytah_Homing_DISABLE:= TRUE;
	ELSIF VystupVytah.IN.PrechodDopravnikaVytahu_OS6 THEN
		Vizu.TL_VystupVytah_Homing_DISABLE:= TRUE;
	ELSIF NOT VystupVytah.MenicZdvihu_FM3.STAV.READY THEN
		Vizu.TL_VystupVytah_Homing_DISABLE:= TRUE;
	ELSE
		Vizu.TL_VystupVytah_Homing_DISABLE:= FALSE;
	END_IF

	//Tlačítka zdvihu výstupného výťahu//
	IF NOT Safety.STAV.ZonaVystupnyVytah_AKTIVNA THEN
		Vizu.TL_VystupVytah_Zdvih_DISABLE:= TRUE;
	ELSIF VystupVytah.RR_Dopravnik_VPRED THEN
		Vizu.TL_VystupVytah_Zdvih_DISABLE:= TRUE;
	ELSIF VystupVytah.RR_Dopravnik_VZAD THEN
		Vizu.TL_VystupVytah_Zdvih_DISABLE:= TRUE;
	ELSIF VystupVytah.STAV.Homing_BUSY THEN
		Vizu.TL_VystupVytah_Zdvih_DISABLE:= TRUE;
	ELSIF VystupVytah.IN.PrechodDopravnikaVytahu_OS6 THEN
		Vizu.TL_VystupVytah_Zdvih_DISABLE:= TRUE;
	ELSIF NOT VystupVytah.MenicZdvihu_FM3.STAV.READY THEN
		Vizu.TL_VystupVytah_Zdvih_DISABLE:= TRUE;
	ELSE
		Vizu.TL_VystupVytah_Zdvih_DISABLE:= FALSE;
	END_IF

	//Tlačítko odparkuj robota//
	IF Linka.STAV.Automat THEN
		Vizu.TL_OdparkujRobota_DISABLE:= TRUE;
	ELSIF NOT Safety.STAV.ZonaBunky_AKTIVNA THEN
		Vizu.TL_OdparkujRobota_DISABLE:= TRUE;
	ELSIF SC_Robot.Step <> 1 THEN
		Vizu.TL_OdparkujRobota_DISABLE:= TRUE;
	ELSIF Safety.STAV.MutingRobota_AKTIVNY THEN
		Vizu.TL_OdparkujRobota_DISABLE:= TRUE;
	ELSIF NOT Robot.KOM_IN.Stav_RezimAUTOMAT THEN
		Vizu.TL_OdparkujRobota_DISABLE:= TRUE;
	ELSE
		Vizu.TL_OdparkujRobota_DISABLE:= FALSE;
	END_IF

	//Tlačítka ovládania bunky v ručnom režime//
	IF Safety.STAV.ZonaBunky_AKTIVNA THEN
		Vizu.TL_BunkyRR_DISABLE:= FALSE;
	ELSE
		Vizu.TL_BunkyRR_DISABLE:= TRUE;
	END_IF

	//Tlačítko presun robota na pozíciu čítania interného štítku//
	IF Linka.STAV.Automat THEN
		Vizu.TL_Robot_CitanieQRkodu_DISABLE:= TRUE;
	ELSIF Robot.RR_PresunPoziciaCitaniaDMkodu THEN
		Vizu.TL_Robot_CitanieQRkodu_DISABLE:= TRUE;
	ELSIF Robot.RR_PresunPoziciaOdobratiaEtikety THEN
		Vizu.TL_Robot_CitanieQRkodu_DISABLE:= TRUE;
	ELSIF NOT Safety.STAV.ZamkyBunky_AKTIVNE THEN
		Vizu.TL_Robot_CitanieQRkodu_DISABLE:= TRUE;
	ELSIF NOT Safety.STAV.ZonaCS_AKTIVNA THEN
		Vizu.TL_Robot_CitanieQRkodu_DISABLE:= TRUE;
	ELSIF NOT Robot.KOM_IN.Stav_RezimAUTOMAT THEN
		Vizu.TL_Robot_CitanieQRkodu_DISABLE:= TRUE;
	ELSIF NOT Safety.STAV.ServisneDvereTlaciarne_AKTIVNE THEN
		Vizu.TL_Robot_CitanieQRkodu_DISABLE:= TRUE;
	ELSIF NOT StoperEtiketovania.IN.SuflikTlaciarne_LS_IS23 OR NOT StoperEtiketovania.IN.SuflikTlaciarne_PS_IS22 THEN
		Vizu.TL_Robot_CitanieQRkodu_DISABLE:= TRUE;
	ELSIF Linka.PAR.Zvoleny_MODEL = '' THEN
		Vizu.TL_Robot_CitanieQRkodu_DISABLE:= TRUE;
	ELSE
		Vizu.TL_Robot_CitanieQRkodu_DISABLE:= FALSE;
	END_IF

	//Tlačítko presun robota na pozíciu čítania zákaznického štítku//
	IF Linka.STAV.Automat THEN
		Vizu.TL_Robot_CitanieDMkodu_DISABLE:= TRUE;
	ELSIF Robot.RR_PresunPoziciaCitaniaQRkodu THEN
		Vizu.TL_Robot_CitanieDMkodu_DISABLE:= TRUE;
	ELSIF Robot.RR_PresunPoziciaOdobratiaEtikety THEN
		Vizu.TL_Robot_CitanieDMkodu_DISABLE:= TRUE;
	ELSIF NOT Safety.STAV.ZamkyBunky_AKTIVNE THEN
		Vizu.TL_Robot_CitanieDMkodu_DISABLE:= TRUE;
	ELSIF NOT Safety.STAV.ZonaCS_AKTIVNA THEN
		Vizu.TL_Robot_CitanieDMkodu_DISABLE:= TRUE;
	ELSIF NOT Robot.KOM_IN.Stav_RezimAUTOMAT THEN
		Vizu.TL_Robot_CitanieDMkodu_DISABLE:= TRUE;
	ELSIF NOT Safety.STAV.ServisneDvereTlaciarne_AKTIVNE THEN
		Vizu.TL_Robot_CitanieDMkodu_DISABLE:= TRUE;
	ELSIF NOT StoperEtiketovania.IN.SuflikTlaciarne_LS_IS23 OR NOT StoperEtiketovania.IN.SuflikTlaciarne_PS_IS22 THEN
		Vizu.TL_Robot_CitanieDMkodu_DISABLE:= TRUE;
	ELSIF Linka.PAR.Zvoleny_MODEL = '' THEN
		Vizu.TL_Robot_CitanieDMkodu_DISABLE:= TRUE;
	ELSE
		Vizu.TL_Robot_CitanieDMkodu_DISABLE:= FALSE;
	END_IF

	//Tlačátko presun robota na pozíciu odobratia etikety z tlačiarne//
	IF Linka.STAV.Automat THEN
		Vizu.TL_Robot_OdoberEtiketu_DISABLE:= TRUE;
	ELSIF Robot.RR_PresunPoziciaCitaniaQRkodu THEN
		Vizu.TL_Robot_OdoberEtiketu_DISABLE:= TRUE;
	ELSIF Robot.RR_PresunPoziciaCitaniaDMkodu THEN
		Vizu.TL_Robot_OdoberEtiketu_DISABLE:= TRUE;
	ELSIF NOT Safety.STAV.ZamkyBunky_AKTIVNE THEN
		Vizu.TL_Robot_OdoberEtiketu_DISABLE:= TRUE;
	ELSIF NOT Safety.STAV.ZonaCS_AKTIVNA THEN
		Vizu.TL_Robot_OdoberEtiketu_DISABLE:= TRUE;
	ELSIF NOT Robot.KOM_IN.Stav_RezimAUTOMAT THEN
		Vizu.TL_Robot_OdoberEtiketu_DISABLE:= TRUE;
	ELSIF NOT Safety.STAV.ServisneDvereTlaciarne_AKTIVNE THEN
		Vizu.TL_Robot_OdoberEtiketu_DISABLE:= TRUE;
	ELSIF NOT StoperEtiketovania.IN.SuflikTlaciarne_LS_IS23 OR NOT StoperEtiketovania.IN.SuflikTlaciarne_PS_IS22 THEN
		Vizu.TL_Robot_OdoberEtiketu_DISABLE:= TRUE;
	ELSIF Linka.PAR.Zvoleny_MODEL = '' THEN
		Vizu.TL_Robot_OdoberEtiketu_DISABLE:= TRUE;
	ELSE
		Vizu.TL_Robot_OdoberEtiketu_DISABLE:= FALSE;
	END_IF

	//Tlačítko ovládania Ionizátora//
	IF NOT VstupVytah.IN.DvereVytahuZatvorene_MS2 THEN
		Vizu.TL_Ovl_Ionizatora_DISABLE:= TRUE;
	ELSE
		Vizu.TL_Ovl_Ionizatora_DISABLE:= FALSE;
	END_IF

	//Ovládanie dverí vstupného výťahu//
	IF NOT Safety.STAV.BarieraVstupVytahu_AKTIVNA THEN
		Vizu.TL_Ovl_DveriVstupVytahu_DISABLE:= TRUE;
	ELSE
		Vizu.TL_Ovl_DveriVstupVytahu_DISABLE:= FALSE;
	END_IF

	//Zadávanie korekcii robota//
	IF OffsetRobota_NazovModelu = '' THEN
		Vizu.ZadavanieKorekciiRobota_DISABLE:= TRUE;
	ELSE
		Vizu.ZadavanieKorekciiRobota_DISABLE:= FALSE;
	END_IF

	//Volby režimov//
	IF Linka.STAV.Automat THEN
		Vizu.VolbyRezimov_DISABLE:= TRUE;
	ELSIF ZvolenaUroven < 20 THEN
		Vizu.VolbyRezimov_DISABLE:= TRUE;
	ELSE
		Vizu.VolbyRezimov_DISABLE:= FALSE;
	END_IF

	//Zadávanie parametrov//
	IF Linka.STAV.Automat THEN
		Vizu.ZmenaParametrov_DISABLE:= TRUE;
	ELSE
		Vizu.ZmenaParametrov_DISABLE:= FALSE;
	END_IF

	//Vypnutie hlásenia koniec pásky alebo etikiet v tlačiarni//
	IF NOT StoperEtiketovania.IN.Tlaciaren_KoniecEtikiet AND NOT StoperEtiketovania.IN.Tlaciaren_KoniecPasky THEN
		Vizu.ZobrazHlasenie_DochadzaPaska:= 1;
	END_IF

	//***********************************************Prepínanie obrázkov súradnicového systému pre zadávanie korekcii robota*******************************************************//
	IF RFID_Hlava_2.PAR.PrecitanyTypPaletky = 'BD1' THEN
		Vizu.IndexSuradnicovehoSystemuPaletky:= 1;
	ELSIF RFID_Hlava_2.PAR.PrecitanyTypPaletky = 'BE1' THEN
		Vizu.IndexSuradnicovehoSystemuPaletky:= 2;
	ELSIF RFID_Hlava_2.PAR.PrecitanyTypPaletky = 'BF1' THEN
		Vizu.IndexSuradnicovehoSystemuPaletky:= 3;
	ELSIF RFID_Hlava_2.PAR.PrecitanyTypPaletky = 'BV1' THEN
		Vizu.IndexSuradnicovehoSystemuPaletky:= 4;
	ELSIF RFID_Hlava_2.PAR.PrecitanyTypPaletky = 'EH1' THEN
		Vizu.IndexSuradnicovehoSystemuPaletky:= 4;
	ELSIF RFID_Hlava_2.PAR.PrecitanyTypPaletky = 'BW1' THEN
		Vizu.IndexSuradnicovehoSystemuPaletky:= 5;
	ELSIF RFID_Hlava_2.PAR.PrecitanyTypPaletky = 'CN1' THEN
		Vizu.IndexSuradnicovehoSystemuPaletky:= 6;
	ELSIF RFID_Hlava_2.PAR.PrecitanyTypPaletky = 'CP1' THEN
		Vizu.IndexSuradnicovehoSystemuPaletky:= 7;
	END_IF

	//***********************************************Zobrazenie stavov ladenia kamery***********************************************//
	//0 - READY.
	//1 - Paletka nieje zacentrovana !!!.
	//2 - Na pozícii etiketovania nie je paletka !!!.
	//3 - Dvere bunky nie su zamknuté !!!
	//4 - Zóna CS nieje aktívna !!!
	//5 - Robot nie je prepnutý do automatického režimu !!!
	//6 - Ukonči automatický režim linky !!!
	//7 - Servisné dvere tlačiarne nie su zatvorené !!!
	//8 - Tlačiareň nie je zaaretovaná !!!
	//9 - Na linke nieje zvolený model !!!

	//Farba//
	//0 - červená
	//1 - zelená

	IF NOT RFID_Hlava_2.STAV.PritomnostCipu THEN
		Vizu.IndexStavuLadenieKamery:= 2;
		Vizu.IndexStavuLadenieKamery_Farba:= 0;
	ELSIF NOT Safety.STAV.ZamkyBunky_AKTIVNE THEN
		Vizu.IndexStavuLadenieKamery:= 3;
		Vizu.IndexStavuLadenieKamery_Farba:= 0;
	ELSIF NOT Safety.STAV.ZonaCS_AKTIVNA THEN
		Vizu.IndexStavuLadenieKamery:= 4;
		Vizu.IndexStavuLadenieKamery_Farba:= 0;
	ELSIF NOT Robot.KOM_IN.Stav_RezimAUTOMAT THEN
		Vizu.IndexStavuLadenieKamery:= 5;
		Vizu.IndexStavuLadenieKamery_Farba:= 0;
	ELSIF Linka.STAV.Automat THEN
		Vizu.IndexStavuLadenieKamery:= 6;
		Vizu.IndexStavuLadenieKamery_Farba:= 0;
	ELSIF NOT Safety.STAV.ServisneDvereTlaciarne_AKTIVNE THEN
		Vizu.IndexStavuLadenieKamery:= 7;
		Vizu.IndexStavuLadenieKamery_Farba:= 0;
	ELSIF NOT StoperEtiketovania.IN.SuflikTlaciarne_LS_IS23 OR NOT StoperEtiketovania.IN.SuflikTlaciarne_PS_IS22 THEN
		Vizu.IndexStavuLadenieKamery:= 8;
		Vizu.IndexStavuLadenieKamery_Farba:= 0;
	ELSIF Linka.PAR.Zvoleny_MODEL = '' THEN
		Vizu.IndexStavuLadenieKamery:= 9;
		Vizu.IndexStavuLadenieKamery_Farba:= 0;
	ELSE
		Vizu.IndexStavuLadenieKamery:= 0;
		Vizu.IndexStavuLadenieKamery_Farba:= 1;
	END_IF

END_PROGRAM

PROGRAM _EXIT
	(* Insert code here *)

END_PROGRAM
```

- Visualisation Logical/HMI/Visu (not shown)

### Program Logical/EthernetovaKomunikacia/EthernetovaKomunikacia (IEC)

#### Main.st - Init, cyclic, exit code
```iecst
PROGRAM _INIT
	(* Insert code here *)

END_PROGRAM

PROGRAM _CYCLIC

	CASE Client.sStep OF

		0://Čakanie na spustenie komunikácie z tlačiarňou//
			IF StoperEtiketovania.OUT.Tlaciaren_VytlacEtiketu THEN
				Tlaciaren.Status.PoruchaOtvoreniaKomunikacie:= FALSE;
				Tlaciaren.Status.PoruchaSpojenia_s_Tlaciarnou:= FALSE;
				Tlaciaren.Status.PoruchaOdoslaniaDat:= FALSE;
				Tlaciaren.Status.PoruchaZatvoreniaKomunikacie:= FALSE;
				Tlaciaren.Status.PoruchaPrijatiaDat:= FALSE;
				Tlaciaren.Status.PrislaSprava_s_Tlaciarne:= FALSE;
				(*strcpy(ADR(Tlaciaren.Data.Sprava_pre_Tlaciaren),ADR(''));*)
				strcpy(ADR(Tlaciaren.Data.Odpoved_s_Tlaciarne),ADR('')); //Vynulovanie premennej typu string
				Client.sStep := 1;
			END_IF

		1: //Otvorenie ethernetovej komunikácie//
			Client.TcpOpen_0.enable := 1;
			Client.TcpOpen_0.pIfAddr := 0;  (* Which Interface to open *)
			Client.TcpOpen_0.port := 9100;  (* Port komunikácie s tlačiarňou *)
			Client.TcpOpen_0.options := 0;
			Client.TcpOpen_0;  (* Call the Function *)

			IF Client.TcpOpen_0.status = 0 THEN  (* TCP port je otvorený *)
				Client.TcpOpen_timeout := 0;
				Client.sStep := 5;
			ELSIF Client.TcpOpen_0.status = ERR_FUB_BUSY THEN  (* TCP port sa otvára *)
				Client.TcpOpen_timeout := Client.TcpOpen_timeout + 1;
				IF Client.TcpOpen_timeout > 50 THEN
					Tlaciaren.Status.PoruchaOtvoreniaKomunikacie:= TRUE;
					Client.TcpOpen_timeout := 0;
					Client.sStep := 40;
				END_IF
					(* Busy *)
			ELSE  (* Goto Error Step *)
				Tlaciaren.Status.PoruchaOtvoreniaKomunikacie:= TRUE;
				Client.TcpOpen_timeout := 0;
				Client.sStep := 100;
			END_IF

		5:
			Client.linger_opt.lLinger := 0; (* linger Time = 0 *)
			Client.linger_opt.lOnOff := 1; (* linger Option ON *)
			Client.TcpIoctl_0.enable := 1;
			Client.TcpIoctl_0.ident := Client.TcpOpen_0.ident; (* Connection Ident from AsTP.TCP_Open *)
			Client.TcpIoctl_0.ioctl := tcpSO_LINGER_SET; (* Set Linger Options *)
			Client.TcpIoctl_0.pData := ADR(Client.linger_opt);
			Client.TcpIoctl_0.datalen := SIZEOF(Client.linger_opt);
			Client.TcpIoctl_0;

			IF Client.TcpIoctl_0.status = 0 THEN  (* TcpIoctl successfull *)
				Client.sStep := 10;
			ELSIF Client.TcpIoctl_0.status = ERR_FUB_BUSY THEN  (* TcpIoctl not finished -> redo *)
				(* Busy *)
			ELSE  (* Goto Error Step *)
				Client.sStep := 100;
			END_IF

		10: //Spojenie s tlačiarňou//
			Client.TcpClient_0.enable := 1;
			Client.TcpClient_0.ident := Client.TcpOpen_0.ident;  (* Connection Ident from AsTCP.TCP_Open *)
			Client.TcpClient_0.portserv := 9100;  (* Port komunikácie s tlačiarňou *)
			Client.TcpClient_0.pServer := ADR('192.168.1.113');  (* Adresa tlačiarne *)
			Client.TcpClient_0;  (* Call the Function*)

			IF Client.TcpClient_0.status = 0 THEN  (* Open ok -> Send Data *)
				Client.TcpClient_timeout := 0;
				Client.sStep := 20;
			ELSIF Client.TcpClient_0.status = ERR_FUB_BUSY THEN  (* TcpClient not finished -> redo *)
				Client.TcpClient_timeout := Client.TcpClient_timeout + 1;
				IF Client.TcpClient_timeout > 50 THEN
					Tlaciaren.Status.PoruchaSpojenia_s_Tlaciarnou:= TRUE;
					Client.TcpClient_timeout := 0;
					Client.sStep := 40;
				END_IF

				(* Busy *)
			ELSIF Client.TcpClient_0.status = tcpERR_INVALID THEN  (* Port error -> Close actual connection, and reopen a new one *)
				Client.TcpClient_timeout := 0;
				Client.sStep := 40;
			ELSE  (* Goto Error Step *)
				Tlaciaren.Status.PoruchaSpojenia_s_Tlaciarnou:= TRUE;
				Client.TcpClient_timeout := 0;
				Client.sStep := 100;
			END_IF

		20: //Poslanie dát do tlačiarne//
			Client.TcpSend_0.enable := 1;
			Client.TcpSend_0.ident := Client.TcpOpen_0.ident;  (* Connection Ident from AsTCP.TCP_Open *)
			Client.TcpSend_0.pData := ADR(Tlaciaren.Data.Sprava_pre_Tlaciaren);  (* Dáta poslané do tlačiarne *)
			Client.TcpSend_0.datalen := SIZEOF(Tlaciaren.Data.Sprava_pre_Tlaciaren);  (* Lenght of data to send *)
			Client.TcpSend_0.flags := 0;
			Client.TcpSend_0;  (* Call the Function*)

			IF Client.TcpSend_0.status = 0 THEN  (* Data was sent sucessfully -> receive data *)
				Client.sStep := 40;
			ELSIF Client.TcpSend_0.status = ERR_FUB_BUSY THEN  (* TcpSend not finished -> redo *)
				(* Busy *)
			ELSIF (Client.TcpSend_0.status = tcpERR_SENTLEN) OR (Client.TcpSend_0.status = tcpERR_NOT_CONNECTED) THEN (* Connection Lost *)
				Client.sStep := 40;
			ELSE  (* Goto Error Step *)
				Tlaciaren.Status.PoruchaOdoslaniaDat:= TRUE;
				Client.sStep := 100;
			END_IF

		30: //Prijatie odpovede s tlačiarne//
			Client.TcpRecv_0.enable := 1;
			Client.TcpRecv_0.ident := Client.TcpOpen_0.ident;  (* Connection Ident from AsTCP.TCP_Open *)
			Client.TcpRecv_0.pData	:= ADR(Tlaciaren.Data.Odpoved_s_Tlaciarne);  (* Dáta poslané z tlačiarne *)
			Client.TcpRecv_0.datamax := SIZEOF(Tlaciaren.Data.Odpoved_s_Tlaciarne);  (* Lenght of data buffer *)
			Client.TcpRecv_0.flags := 0;
			Client.TcpRecv_0;  (* Call the Function*)

			IF Client.TcpRecv_0.status = 0 THEN  (* Data was received sucessfully -> Send next packet *)
				Tlaciaren.Status.PrislaSprava_s_Tlaciarne:= TRUE;
				Client.recv_timeout := 0;
				Client.sStep := 40;
			ELSIF Client.TcpRecv_0.status = tcpERR_NO_DATA THEN  (* No data received - wait *)
				Client.recv_timeout := Client.recv_timeout + 1;
				IF Client.recv_timeout > 50 THEN
					Client.recv_timeout := 0;
					Client.sStep := 40;
				END_IF
				(* No Data received *)
			ELSIF Client.TcpRecv_0.status = ERR_FUB_BUSY THEN  (* TcpRecv not finished -> redo *)
				(* Busy *)
			ELSIF Client.TcpRecv_0.status = tcpERR_NOT_CONNECTED THEN (* Connection Lost *)
				Client.recv_timeout := 0;
				Client.sStep := 40;
			ELSE  (* Goto Error Step *)
				Tlaciaren.Status.PoruchaPrijatiaDat:= TRUE;
				Client.recv_timeout := 0;
				Client.sStep := 100;
			END_IF

		40: //Zatvorenie ethernetovej komunikácie//
			Client.TcpClose_0.enable := 1;
			Client.TcpClose_0.ident := Client.TcpOpen_0.ident;  (* Connection Ident from AsTCP.TCP_Open *)
			Client.TcpClose_0.how := 0;
			Client.TcpClose_0;  (* Call the Function*)

			IF Client.TcpClose_0.status = 0 THEN  (* Close sucessfull -> Reopen the interface *)
				Client.sStep := 100;
			ELSIF Client.TcpClose_0.status = ERR_FUB_BUSY THEN  (* TcpClose not finished -> redo *)
				(* Busy *)
			ELSE  (* Goto Error Step *)
				Tlaciaren.Status.PoruchaZatvoreniaKomunikacie:= TRUE;
				Client.sStep := 100;
			END_IF

		100: //Ukončenie komunikácie s tlačiarňou//
			StoperEtiketovania.OUT.Tlaciaren_VytlacEtiketu:= FALSE;
			Tlaciaren.Commands.PosliSpravu:= FALSE;
			Client.sStep := 0;

	END_CASE

END_PROGRAM

PROGRAM _EXIT
	(* Insert code here *)

END_PROGRAM
```

### DatumCasGlobal.var
```iecst
VAR
	PLC_Cas : PLC_Cas_typ;
	PLC_Datum : PLC_Datum_typ;
	Sekunda_STR : STRING[2];
	Minuta_STR : STRING[2];
	Hodina_STR : STRING[2];
	Den_STR : STRING[2];
	Mesiac_STR : STRING[2];
	Rok_STR_4_Znaky : STRING[4];
	Rok_STR_2_Znaky : STRING[2];
	DTSetTime_0 : DTSetTime;
	DTGetTime_0 : DTGetTime;
END_VAR
```

### DatumCasGlobal.typ
```iecst
TYPE
	PLC_Cas_typ : 	STRUCT
		Sekundy : USINT;
		Minuty : USINT;
		Hodiny : USINT;
	END_STRUCT;
	PLC_Datum_typ : 	STRUCT
		Den : USINT;
		Mesiac : USINT;
		Rok : UINT;
	END_STRUCT;
END_TYPE
```

### Program Logical/DatumCasPLC/DatumCasPLC (IEC)

#### Main.st - Init, cyclic, exit code
```iecst
PROGRAM _INIT
	(* Insert code here *)

END_PROGRAM

PROGRAM _CYCLIC

	//Vyčítavanie systémového času//
	DTGetTime_1.enable:= TRUE;
	DTGetTime_1();
	DT_TO_DTStructure(DTGetTime_1.DT1,ADR(PLC_DatumCas));

	PLC_Cas.Sekundy:= PLC_DatumCas.second;
	PLC_Cas.Minuty:= PLC_DatumCas.minute;
	PLC_Cas.Hodiny:= PLC_DatumCas.hour;

	PLC_Datum.Den:= PLC_DatumCas.day;
	PLC_Datum.Mesiac:= PLC_DatumCas.month;
	PLC_Datum.Rok:= PLC_DatumCas.year;

	//Prevod času na String//
	//Sekundy//
	IF PLC_Cas.Sekundy < 10 THEN
		Sekundy_String:= USINT_TO_STRING(PLC_Cas.Sekundy);
		Sekunda_STR:= '0';
		brsstrcat(ADR(Sekunda_STR),ADR(Sekundy_String));
	ELSE
		Sekunda_STR:= USINT_TO_STRING(PLC_Cas.Sekundy);
	END_IF

	//Minuty//
	IF PLC_Cas.Minuty < 10 THEN
		Minuty_String:= USINT_TO_STRING(PLC_Cas.Minuty);
		Minuta_STR:= '0';
		brsstrcat(ADR(Minuta_STR),ADR(Minuty_String));
	ELSE
		Minuta_STR:= USINT_TO_STRING(PLC_Cas.Minuty);
	END_IF

	//Hodiny//
	IF PLC_Cas.Hodiny < 10 THEN
		Hodiny_String:= USINT_TO_STRING(PLC_Cas.Hodiny);
		Hodina_STR:= '0';
		brsstrcat(ADR(Hodina_STR),ADR(Hodiny_String));
	ELSE
		Hodina_STR:= USINT_TO_STRING(PLC_Cas.Hodiny);
	END_IF

	//Prevod dátumu na String//
	//Deň//
	IF PLC_Datum.Den < 10 THEN
		Den_String:= USINT_TO_STRING(PLC_Datum.Den);
		Den_STR:= '0';
		brsstrcat(ADR(Den_STR),ADR(Den_String));
	ELSE
		Den_STR:= USINT_TO_STRING(PLC_Datum.Den);
	END_IF

	//Masiac//
	IF PLC_Datum.Mesiac < 10 THEN
		Mesiac_String:= USINT_TO_STRING(PLC_Datum.Mesiac);
		Mesiac_STR:= '0';
		brsstrcat(ADR(Mesiac_STR),ADR(Mesiac_String));
	ELSE
		Mesiac_STR:= USINT_TO_STRING(PLC_Datum.Mesiac);
	END_IF

	//Rok - 4 znaky//
	Rok_STR_4_Znaky:= UINT_TO_STRING(PLC_Datum.Rok);

	//Rok - posledné 2 znaky//
	length := brsstrlen(ADR(Rok_STR_4_Znaky)); //Zistí počet znakov//

	IF length >= 4 THEN
		brsmemcpy(ADR(PoleUSINT),ADR(Rok_STR_4_Znaky),SIZEOF(Rok_STR_4_Znaky));
		i := PoleUSINT[length-2]; //Vyčítanie predposledného znaku//
		brsstrcpy(ADR(DvaZnaky),ADR(i));
		i := PoleUSINT[length-1]; //Vyčítanie posledneho znaku//
		brsstrcat(ADR(DvaZnaky),ADR(i));
	END_IF

	Rok_STR_2_Znaky:= DvaZnaky;

END_PROGRAM

PROGRAM _EXIT
	(* Insert code here *)

END_PROGRAM
```

#### Variables.var - Local variables
```iecst
VAR
	PLC_DatumCas : DTStructure;
	DTGetTime_1 : DTGetTime;
	Sekundy_String : STRING[2];
	Minuty_String : STRING[2];
	Hodiny_String : STRING[2];
	Den_String : STRING[2];
	Mesiac_String : STRING[2];
	length : UDINT;
	PoleUSINT : ARRAY[0..3] OF USINT;
	i : USINT;
	DvaZnaky : STRING[2];
END_VAR
```

### Program Logical/Blikace/Blikanie100ms (IEC)

#### Blikanie100ms.st - Init, cyclic, exit code
```iecst
PROGRAM _INIT
	(* Insert code here *)

END_PROGRAM

PROGRAM _CYCLIC

	IF NOT Blikac100ms THEN
		Blikac100ms:= TRUE;
	ELSE
		Blikac100ms:= FALSE;
	END_IF

END_PROGRAM

PROGRAM _EXIT
	(* Insert code here *)

END_PROGRAM
```

### Program Logical/Blikace/Blikanie200ms (IEC)

#### Blikanie200ms.st - Init, cyclic, exit code
```iecst
PROGRAM _INIT
	(* Insert code here *)

END_PROGRAM

PROGRAM _CYCLIC

	IF NOT Blikac200ms THEN
		Blikac200ms:= TRUE;
	ELSE
		Blikac200ms:= FALSE;
	END_IF

END_PROGRAM

PROGRAM _EXIT
	(* Insert code here *)

END_PROGRAM
```

### Program Logical/Blikace/Blikanie500ms (IEC)

#### Blikanie500ms.st - Init, cyclic, exit code
```iecst
PROGRAM _INIT
	(* Insert code here *)

END_PROGRAM

PROGRAM _CYCLIC
	IF NOT Blikac500ms THEN
		Blikac500ms:= TRUE;
	ELSE
		Blikac500ms:= FALSE;
	END_IF

END_PROGRAM

PROGRAM _EXIT
	(* Insert code here *)

END_PROGRAM
```

### Program Logical/Blikace/Blikanie1s (IEC)

#### Blikanie1s.st - Init, cyclic, exit code
```iecst
PROGRAM _INIT
	(* Insert code here *)

END_PROGRAM

PROGRAM _CYCLIC
	IF NOT Blikac1s THEN
		Blikac1s:= TRUE;
		Pocitadlo:= Pocitadlo + 1;
		IF Pocitadlo > 300 THEN
			Pocitadlo:= 0;
		END_IF
	ELSE
		Blikac1s:= FALSE;
	END_IF

END_PROGRAM

PROGRAM _EXIT
	(* Insert code here *)

END_PROGRAM
```

### Program Logical/Receptury/Receptury (IEC)

#### Main.st - Init, cyclic, exit code
```iecst
PROGRAM _INIT

END_PROGRAM

PROGRAM _CYCLIC

	//Načítanie receptur pri prvom spustení//
	IF EDGEPOS(Safety.STAV.SafetyPLC_Nabehlo = TRUE) THEN
		MpRecipeXml_1.Load:= TRUE;
	END_IF

	//Načítanie receptur z pamäte//
	IF MpRecipeXml_1.Load AND (MpRecipeXml_1.CommandDone OR MpRecipeXml_1.Error) THEN
		MpRecipeXml_1.Load:= FALSE;
		old_i:= 1;
		i:= 0;
		IndexZoznam:= 0;
	END_IF

	//Konfigurácia receptur//
	MpRecipeXml_1.MpLink:= ADR(gRecipeXmlLink);  //takto sa menuje mapp komponenta v configurating view//
	MpRecipeXml_1.Enable:= TRUE;
	MpRecipeXml_1.Category:= ADR('RECEPTURY');
	MpRecipeXml_1.DeviceName:= ADR('HDD');  //Názov media, kde sa budú receptury ukladat//
	MpRecipeXml_1.FileName:= ADR('UlozeneReceptury'); //Názov súboru do ktorého sa receptúry uložia//
	MpRecipeXml_1();

	MpRecipeRegPar_1.MpLink:= ADR(gRecipeXmlLink);
	MpRecipeRegPar_1.Enable:= TRUE;
	MpRecipeRegPar_1.Category:= ADR('RECEPTURY');
	MpRecipeRegPar_1.PVName:= ADR('Receptura'); //Názov premenné, kde je vytvorená štruktura dat pre receptury//
	MpRecipeRegPar_1();

	//Zobrazenie názvou receptúr//
	FOR IndexZoznam:=0 TO 150 BY 1 DO
		ZoznamReceptur[IndexZoznam]:= Receptura[IndexZoznam].NazovModelu;
	END_FOR

	//Posun indexu//
	IF MoveUP THEN
		IF i< 150 THEN
			i:= i+1;
		END_IF
		MoveUP:= FALSE;
	END_IF

	IF MoveDown THEN
		IF i>0 THEN
			i:= i-1;
		END_IF
		MoveDown:= FALSE;
	END_IF

	//Posun indexu po stranách//
	IF MoveUP_Page THEN
		IF i< (150 - 7) THEN
			i:= i+7;
		END_IF
		MoveUP_Page:= FALSE;
	END_IF

	IF MoveDown_Page THEN
		IF i>(0+7) THEN
			i:= i-7;
		END_IF
		MoveDown_Page:= FALSE;
	END_IF

	//Listovanie v uložených recepturach//
	IF old_i <> i THEN
		NazovModelu:= Receptura[i].NazovModelu;
		TypPaletky:= Receptura[i].TypPaletky;
		Robot_CisloProgramu:= Receptura[i].Robot_CisloProgramu;
		Kamera_CisloProgramu_QRkod:= Receptura[i].Kamera_CisloProgramuQRkod;
		Kamera_CisloProgramu_DMkod:= Receptura[i].Kamera_CisloProgramuDMkod;
		RychlostDopravnikaPriCisteni:= Receptura[i].RychlostDopravnikaPriCisteni;
		old_i:= i;
	END_IF

	//Vymazanie receptury//
	IF VymazRecepturu THEN
		RecipeVymazanie_DONE:= FALSE;
		Receptura[i].NazovModelu:= '';
		Receptura[i].TypPaletky:= '';
		Receptura[i].Robot_CisloProgramu:= 0;
		Receptura[i].Kamera_CisloProgramuQRkod:= 0;
		Receptura[i].Kamera_CisloProgramuDMkod:= 0;
		Receptura[i].RychlostDopravnikaPriCisteni:= 0;
		Receptura[i].Robot_PozLepenia_OffsetX:= 0;
		Receptura[i].Robot_PozLepenia_OffsetY:= 0;
		Receptura[i].Robot_PozLepenia_OffsetZ:= 0;
		MpRecipeXml_1.Save:= TRUE;
		RecipeVymazanie_DONE:= TRUE;
		VymazRecepturu:= FALSE;
	END_IF

	//Prepísanie receptury//
	IF PrepisRecepturu THEN
		RecipePrepis_DONE:= FALSE;
		Receptura[i].NazovModelu:= NazovModelu;
		Receptura[i].TypPaletky:= TypPaletky;
		Receptura[i].Robot_CisloProgramu:= Robot_CisloProgramu;
		Receptura[i].Kamera_CisloProgramuQRkod:= Kamera_CisloProgramu_QRkod;
		Receptura[i].Kamera_CisloProgramuDMkod:= Kamera_CisloProgramu_DMkod;
		Receptura[i].RychlostDopravnikaPriCisteni:= RychlostDopravnikaPriCisteni;
		MpRecipeXml_1.Save:= TRUE;
		RecipePrepis_DONE:= TRUE;
		PrepisRecepturu:= FALSE;
	END_IF

	//Uloženie receptury//
	IF UlozRecepturu THEN
		RecipeZapis_DONE:= FALSE;
		FOR a:= 0 TO 150 BY 1 DO
			IF Receptura[a].NazovModelu = NazovModelu AND NOT RecipeZapis_DONE THEN
				Receptura[a].TypPaletky:= TypPaletky;
				Receptura[a].Robot_CisloProgramu:= Robot_CisloProgramu;
				Receptura[a].Kamera_CisloProgramuQRkod:= Kamera_CisloProgramu_QRkod;
				Receptura[a].Kamera_CisloProgramuDMkod:= Kamera_CisloProgramu_DMkod;
				Receptura[a].RychlostDopravnikaPriCisteni:= RychlostDopravnikaPriCisteni;
				MpRecipeXml_1.Save:= TRUE;
				RecipeZapis_DONE:= TRUE;
			ELSIF Receptura[a].NazovModelu = '' AND NOT RecipeZapis_DONE THEN
				Receptura[a].NazovModelu:= NazovModelu;
				Receptura[a].TypPaletky:= TypPaletky;
				Receptura[a].Robot_CisloProgramu:= Robot_CisloProgramu;
				Receptura[a].Kamera_CisloProgramuQRkod:= Kamera_CisloProgramu_QRkod;
				Receptura[a].Kamera_CisloProgramuDMkod:= Kamera_CisloProgramu_DMkod;
				Receptura[a].RychlostDopravnikaPriCisteni:= RychlostDopravnikaPriCisteni;
				MpRecipeXml_1.Save:= TRUE;
				RecipeZapis_DONE:= TRUE;
			END_IF
		END_FOR
		UlozRecepturu:= FALSE;
	END_IF

	IF MpRecipeXml_1.CommandDone THEN
		MpRecipeXml_1.Save:= FALSE;
	END_IF

	//Uloženie korekcii robota//
	IF UlozKorekcieRobota THEN
		UlozenieKorekcii_DONE:= FALSE;
		FOR b:= 0 TO 150 BY 1 DO
			IF Receptura[b].NazovModelu = OffsetRobota_NazovModelu AND NOT UlozenieKorekcii_DONE THEN
				Receptura[b].Robot_PozLepenia_OffsetX:= Linka.PAR.Zvolena_PozLepenia_OffsetX;
				Receptura[b].Robot_PozLepenia_OffsetY:= Linka.PAR.Zvolena_PozLepenia_OffsetY;
				Receptura[b].Robot_PozLepenia_OffsetZ:= Linka.PAR.Zvolena_PozLepenia_OffsetZ;
				MpRecipeXml_1.Save:= TRUE;
				UlozenieKorekcii_DONE:= TRUE;
			END_IF
		END_FOR
		UlozKorekcieRobota:= FALSE;
	END_IF

	//Nacitanie korekcii robota//
	IF NacitajKorekcieRobota THEN
		NacitanieKorekcii_DONE:= FALSE;
		FOR c:= 0 TO 150 BY 1 DO
			IF Receptura[c].NazovModelu = OffsetRobota_NazovModelu AND NOT NacitanieKorekcii_DONE THEN
				Linka.PAR.Zvolena_PozLepenia_OffsetX:= Receptura[c].Robot_PozLepenia_OffsetX;
				Linka.PAR.Zvolena_PozLepenia_OffsetY:= Receptura[c].Robot_PozLepenia_OffsetY;
				Linka.PAR.Zvolena_PozLepenia_OffsetZ:= Receptura[c].Robot_PozLepenia_OffsetZ;
				NacitanieKorekcii_DONE:= TRUE;
			END_IF
		END_FOR
		NacitajKorekcieRobota:= FALSE;
	END_IF

	//Načitanie receptur do premenných//
	IF NacitajRecepturu THEN
		Linka.PAR.Zvoleny_TypPaletky:= Receptura[Linka.PAR.IndexZvoleneReceptury].TypPaletky;
		Linka.PAR.Zvolene_CisloProgramuRobota:= Receptura[Linka.PAR.IndexZvoleneReceptury].Robot_CisloProgramu;
		Linka.PAR.Zvolene_KamCisloProg_QRkod:= Receptura[Linka.PAR.IndexZvoleneReceptury].Kamera_CisloProgramuQRkod;
		Linka.PAR.Zvolene_KamCisloProg_DMkod:= Receptura[Linka.PAR.IndexZvoleneReceptury].Kamera_CisloProgramuDMkod;
		Linka.PAR.Zvolena_RychlostDopravPriCisteni:= Receptura[Linka.PAR.IndexZvoleneReceptury].RychlostDopravnikaPriCisteni;
		NacitajRecepturu:= FALSE;
	END_IF

END_PROGRAM

PROGRAM _EXIT
	(* Insert code here *)

END_PROGRAM
```

#### Variables.var - Local variables
```iecst
VAR
	MpRecipeUI_0 : MpRecipeUI;
	UISetup : MpRecipeUISetupType;
	UIConnect : MpRecipeUIConnectType := (0);
	i : UINT;
	old_i : UINT;
	IndexZoznam : UINT;
	MoveUP : BOOL;
	MoveDown : BOOL;
	MoveUP_Page : BOOL;
	MoveDown_Page : BOOL;
	a : UINT := 0;
	RecipeZapis_DONE : BOOL;
	RecipeVymazanie_DONE : BOOL := FALSE;
	RecipePrepis_DONE : BOOL := FALSE;
	b : UINT := 0;
	c : UINT := 0;
	d : UINT := 0;
	e : UINT := 0;
END_VAR
```

### Program Logical/PrihlasovaciSystem/PrihlasovaciSystem (IEC)

#### Main.st - Init, cyclic, exit code
```iecst
PROGRAM _INIT
	MpRecipeXml_2.Load:= TRUE;
	ZvolenyUzivatel:= '';
	ZvolenaUroven:= 0;
	TP_ZobrazPopUpPrihlasenie:=1;

END_PROGRAM

PROGRAM _CYCLIC

	//Volanie funkcie SequenceControl//
	SequenceControl(SC:= SC_Uzivatelia);

	//Načítanie receptur z pamäte//
	IF MpRecipeXml_2.Load AND (MpRecipeXml_2.CommandDone OR MpRecipeXml_2.Error) THEN
		MpRecipeXml_2.Load:= FALSE;
		old_a:= 1;
		i:= 0;
		IndexZoznam:= 0;
	END_IF

	//Konfigurácia receptur//
	MpRecipeXml_2.MpLink:= ADR(gUzivatelXmlLink);  //takto sa menuje mapp komponenta v configurating view//
	MpRecipeXml_2.Enable:= TRUE;
	MpRecipeXml_2.Category:= ADR('UZIVATELIA');
	MpRecipeXml_2.Category:= ADR(strCategory);
	MpRecipeXml_2.DeviceName:= ADR('HDD');  //Názov media, kde sa budú receptury ukladat//
	MpRecipeXml_2.FileName:= ADR('UlozenyUzivatel'); //Názov súboru do ktorého sa receptúry uložia//
	MpRecipeXml_2();

	MpRecipeRegPar_2.MpLink:= ADR(gUzivatelXmlLink);
	MpRecipeRegPar_2.Enable:= TRUE;
	MpRecipeRegPar_2.Category:= ADR('UZIVATELIA');
	MpRecipeRegPar_2.PVName:= ADR('Uzivatel'); //Názov premenné, kde je vytvorená štruktura dat pre receptury//
	MpRecipeRegPar_2();

	//Zobrazenie názvou receptúr//
	FOR IndexZoznam:=0 TO 50 BY 1 DO
		ZoznamUzivatelov[IndexZoznam]:= Uzivatel[IndexZoznam].Meno;
	END_FOR

	//Posun indexu//
	IF MoveUP THEN
		IF i< 50 THEN
			i:= i+1;
		END_IF
		MoveUP:= FALSE;
	END_IF

	IF MoveDown THEN
		IF i>0 THEN
			i:= i-1;
		END_IF
		MoveDown:= FALSE;
	END_IF

	//Listovanie v uložených uživateloch//
	IF old_a <> i AND i >= 0 AND i <= 50 THEN
		MenoUzivatela:= Uzivatel[i].Meno;
		HesloUzivatela:= '*****';
		UrovenUzivatela:= Uzivatel[i].UrovenUzivatela;
		old_a:= i;
	END_IF

	//Automatické odhlásenie uživatela//

	IF ZvolenaUroven > 0 AND ZvolenaUroven < 100 AND Vizu.CisloAktualnejObrazovky = 2 THEN
		CasAutomOdhlaseniaUzivatela.IN:= TRUE;
	ELSE
		CasAutomOdhlaseniaUzivatela.IN:= FALSE;
	END_IF

	IF CasAutomOdhlaseniaUzivatela.Q AND SC_Uzivatelia.Step = 1 THEN
		OdhlasUzivatela:= TRUE;
	END_IF

	CasAutomOdhlaseniaUzivatela.PT:= T#5M;
	CasAutomOdhlaseniaUzivatela();

	//Prihlasovanie//
	CASE SC_Uzivatelia.Step OF

		0://Vynulovanie uživatela//
			SC_Uzivatelia.StepName:= '0 - Nulovanie';
			UlozUzivatelov:= FALSE;
			PrihlasUzivatela:= FALSE;
			VymazUzivatela:= FALSE;
			OdhlasUzivatela:= FALSE;
			MpRecipeXml_2.Save:= FALSE;
			b:= 0;
			c:= 0;
			d:= 0;
			UzivatelNajdeny:= FALSE;
			UzivatelUlozeny:= FALSE;
			SC_Uzivatelia.ResetStep:= TRUE;
			SC_Uzivatelia.Step:= 1;

		1://Rozhodnutie o činnosti//
			SC_Uzivatelia.StepName:= '1 - Rozhodnutie o cinnosti';
			IF UlozUzivatelov THEN
				SC_Uzivatelia.Step:= 10;
			ELSIF PrihlasUzivatela THEN
				SC_Uzivatelia.Step:= 20;
			ELSIF OdhlasUzivatela THEN
				SC_Uzivatelia.Step:= 30;
			ELSIF VymazUzivatela THEN
				SC_Uzivatelia.Step:= 40;
			END_IF

		10://Ulozenie uzivatela//
			SC_Uzivatelia.StepName:= '10 - Ulozenie uzivatela - hladanie existujuceho uzivatela';
			IF MenoUzivatela <> '' AND HesloUzivatela <> '' AND HesloUzivatela <> '*****' THEN
				FOR c:= 0 TO 50 BY 1 DO
					IF Uzivatel[c].Meno = MenoUzivatela AND NOT UzivatelUlozeny THEN
						Uzivatel[c].Heslo:= HesloUzivatela;
						Uzivatel[c].UrovenUzivatela:= UrovenUzivatela;
						MpRecipeXml_2.Save:= TRUE;
						UzivatelUlozeny:= TRUE;
					END_IF
				END_FOR
			ELSE
				SC_Uzivatelia.ResetStep:= TRUE;
				SC_Uzivatelia.Step:= 0;
			END_IF

			IF UzivatelUlozeny AND MpRecipeXml_2.CommandDone THEN
				MpRecipeXml_2.Save:= FALSE;
				SC_Uzivatelia.ResetStep:= TRUE;
				SC_Uzivatelia.Step:= 0;
			ELSIF NOT UzivatelUlozeny THEN
				SC_Uzivatelia.ResetStep:= TRUE;
				SC_Uzivatelia.Step:= 11;
			END_IF

		11:
			//Ulozenie uzivatela//
			SC_Uzivatelia.StepName:= '10 - Ulozenie uzivatela - ulozenie na prve prazdne miesto';

			FOR d:= 0 TO 50 BY 1 DO
				IF Uzivatel[d].Meno = '' AND NOT UzivatelUlozeny THEN
					Uzivatel[d].Meno:= MenoUzivatela;
					Uzivatel[d].Heslo:= HesloUzivatela;
					Uzivatel[d].UrovenUzivatela:= UrovenUzivatela;
					MpRecipeXml_2.Save:= TRUE;
					UzivatelUlozeny:= TRUE;
				END_IF
			END_FOR

			IF UzivatelUlozeny AND MpRecipeXml_2.CommandDone THEN
				MpRecipeXml_2.Save:= FALSE;
				SC_Uzivatelia.ResetStep:= TRUE;
				SC_Uzivatelia.Step:= 0;
			ELSIF NOT UzivatelUlozeny THEN
				SC_Uzivatelia.ResetStep:= TRUE;
				SC_Uzivatelia.Step:= 0;
			END_IF

		20://Čakanie na prihlásenie uživatela//
			SC_Uzivatelia.StepName:= '20 - Kontrola prazdneho uzivatela';
			IF ZadaneMenoUzivatela <> '' AND ZadaneHesloUzivatela <> '' THEN
				SC_Uzivatelia.ResetStep:= TRUE;
				SC_Uzivatelia.Step:= 21;
			ELSE
				ZadaneHesloUzivatela:= '';
				SC_Uzivatelia.ResetStep:= TRUE;
				SC_Uzivatelia.Step:= 0;
			END_IF

		21://Kontrola prihláseného uživatela//
			SC_Uzivatelia.StepName:= '21 - Kontrola prihláseného uzivatela';
			FOR b:= 0 TO 50 BY 1 DO
				IF Uzivatel[b].Meno = ZadaneMenoUzivatela AND Uzivatel[b].Heslo = ZadaneHesloUzivatela AND NOT UzivatelNajdeny THEN
					ZvolenyUzivatel:= Uzivatel[b].Meno;
					ZvolenaUroven:= Uzivatel[b].UrovenUzivatela;
					ZadaneHesloUzivatela:= '';
					TP_ZobrazPopUpPrihlasenie:= 1;
					UzivatelNajdeny:= TRUE;
				ELSIF ZadaneMenoUzivatela = 'DesignMP' AND ZadaneHesloUzivatela = 'vlmardo'	AND NOT UzivatelNajdeny THEN
					ZvolenyUzivatel:= 'DesignMP';
					ZvolenaUroven:= 100;
					ZadaneHesloUzivatela:= '';
					TP_ZobrazPopUpPrihlasenie:= 1;
					UzivatelNajdeny:= TRUE;
				END_IF
			END_FOR
			(*ZadaneMenoUzivatela:= '';*)
			ZadaneHesloUzivatela:= '';
			SC_Uzivatelia.ResetStep:= TRUE;
			SC_Uzivatelia.Step:= 0;

		30://Odhlásenie uživatela//
			SC_Uzivatelia.StepName:= '30 - Odhlasenie uzivatela';
			ZvolenyUzivatel:= '';
			ZvolenaUroven:= 0;
			SC_Uzivatelia.ResetStep:= TRUE;
			SC_Uzivatelia.Step:= 0;

		40://Vymazanie uživatela//
			SC_Uzivatelia.StepName:= '40 - Vymazanie uzivatela';
			Uzivatel[i].Meno:= '';
			Uzivatel[i].Heslo:= '';
			Uzivatel[i].UrovenUzivatela:= 0;
			MpRecipeXml_2.Save:= TRUE;
			IF MpRecipeXml_2.CommandDone THEN
				SC_Uzivatelia.ResetStep:= TRUE;
				SC_Uzivatelia.Step:= 0;
			END_IF

	END_CASE

END_PROGRAM

PROGRAM _EXIT
	(* Insert code here *)

END_PROGRAM
```

#### Variables.var - Local variables
```iecst
VAR
	strCategory : STRING[80];
	MpRecipeUI_1 : MpRecipeUI;
	UISetup : MpRecipeUISetupType;
	UIConnect : MpRecipeUIConnectType := (0);
	i : INT := 0;
	a : INT;
	old_a : INT := 0;
	MoveUP : BOOL;
	MoveDown : BOOL;
	IndexZoznam : INT;
	b : INT;
	c : INT := 0;
	d : INT := 0;
	CasOdhlaseniaUzivatela : TON;
	UzivatelNajdeny : BOOL := 0;
	UzivatelUlozeny : BOOL := FALSE;
	CasAutomOdhlaseniaUzivatela : TON := (0);
END_VAR
```

### Program Logical/RemanentnePremenne/RemanentnePremenne (IEC)

#### Main.st - Init, cyclic, exit code
```iecst
PROGRAM _INIT
	(* Insert code here *)

END_PROGRAM

PROGRAM _CYCLIC
	RemPremenne;

	//Načítanie premenných pri prvom spustení//
	IF EDGEPOS(Safety.STAV.SafetyPLC_Nabehlo) THEN
		NacitajPremenne:= TRUE;
	END_IF

	//Načítanie premenných z pamäte//
	IF NacitajPremenne THEN
		MpRecipeXml_0.Load:= TRUE;
		NacitajPremenne:= FALSE;
	END_IF

	IF MpRecipeXml_0.Load AND (MpRecipeXml_0.CommandDone OR MpRecipeXml_0.Error) THEN
		MpRecipeXml_0.Load:= FALSE;
	END_IF

	//Konfigurácia premenných//
	MpRecipeXml_0.MpLink:= ADR(gRemPremenne);  //takto sa menuje mapp komponenta v configurating view//
	MpRecipeXml_0.Enable:= TRUE;
	MpRecipeXml_0.Category:= ADR('PREMENNE');
	MpRecipeXml_0.DeviceName:= ADR('HDD');  //Názov media, kde sa budú receptury ukladat//
	MpRecipeXml_0.FileName:= ADR('RemPremenne'); //Názov súboru do ktorého sa receptúry uložia//
	MpRecipeXml_0();

	MpRecipeRegPar_0.MpLink:= ADR(gRemPremenne);
	MpRecipeRegPar_0.Enable:= TRUE;
	MpRecipeRegPar_0.Category:= ADR('PREMENNE');
	MpRecipeRegPar_0.PVName:= ADR('RemPremenne'); //Názov premenné, kde je vytvorená štruktura dat premennych//
	MpRecipeRegPar_0();

	//Uloženie premenných//
	IF UlozPremenne THEN
		MpRecipeXml_0.Save:= TRUE;
		UlozPremenne:= FALSE;
	END_IF

	IF MpRecipeXml_0.Save AND (MpRecipeXml_0.CommandDone OR MpRecipeXml_0.Error) THEN
		MpRecipeXml_0.Save:= FALSE;
	END_IF

END_PROGRAM

PROGRAM _EXIT
	(* Insert code here *)

END_PROGRAM
```

#### Variables.var - Local variables
```iecst
VAR
	UISetup : MpRecipeUISetupType;
	UIConnect : MpRecipeUIConnectType := (0);
END_VAR
```

### Poznamky.txt
```
***************FTP**************************
login - admin
heslo - vlmardo

*************Safety*************************
heslo - vlmardo

************Adresy frekvenčných meničov na CANopen*****************
FM1 Dopravník čistenia - 32
FM2 Vstupný výtah - 34
FM3 Vystupny výtah - 36

****************Uroveň Design MP************************************
Meno: DesignMP
Heslo: vlmardo

***************Uloženie typu a čísla paletky na RFID čip************
Zadame číslo paletky + oddelovací znak (;) + typ paletky
Napr:  1;BV1

****************VPN**********************************
Pripojenie na HMI - 192.168.1.110:5900
Pripojenie na počítač kde sú kamery - 192.168.1.114  - Heslo je Tester123

***************FTP kamery*****************************
```
